  Call Extruder(68.03550)
  MoveL 3349 to (-35.61, 39.11, 59.84) mm, rotated rx -180 ry 0 rz 180 deg; joints [-168.693, 58.392, -72.558, 168.348, 76.115, 2.833]
  MoveL 3350 to (-35.61, 39.11, 59.84) mm, rotated rx -180 ry 0 rz 180 deg; joints [-168.693, 58.392, -72.558, 168.348, 76.115, 2.833]
  Call Extruder(68.23307)
  MoveL 3351 to (-35.35, 38.9, 59.84) mm, rotated rx -180 ry 0 rz 180 deg; joints [-168.739, 58.372, -72.572, 168.394, 76.079, 2.829]
  Call Extruder(68.56709)
  MoveL 3352 to (-34.9, 38.57, 59.84) mm, rotated rx -180 ry 0 rz -180 deg; joints [-168.806, 58.336, -72.595, 168.46, 76.017, 2.824]
  MoveL 3353 to (-34.9, 38.57, 59.84) mm, rotated rx -180 ry 0 rz -180 deg; joints [-168.806, 58.336, -72.595, 168.46, 76.017, 2.824]
  Call Extruder(68.89992)
  MoveL 3354 to (-34.45, 38.24, 59.84) mm, rotated rx -180 ry 0 rz -180 deg; joints [-168.874, 58.3, -72.619, 168.527, 75.955, 2.82]
  MoveL 3355 to (-34.45, 38.24, 59.84) mm, rotated rx -180 ry 0 rz -180 deg; joints [-168.874, 58.3, -72.619, 168.527, 75.955, 2.82]
  Call Extruder(69.07917)
  MoveL 3356 to (-34.21, 38.06, 59.84) mm, rotated rx -180 ry 0 rz 180 deg; joints [-168.91, 58.28, -72.632, 168.562, 75.922, 2.817]
  MoveL 3357 to (-34.21, 38.06, 59.84) mm, rotated rx -180 ry 0 rz 180 deg; joints [-168.91, 58.28, -72.632, 168.562, 75.922, 2.817]
  Call Extruder(69.28728)
  MoveL 3358 to (-33.9, 37.89, 59.84) mm, rotated rx -180 ry 0 rz 180 deg; joints [-168.944, 58.257, -72.647, 168.595, 75.882, 2.817]
  MoveL 3359 to (-33.9, 37.89, 59.84) mm, rotated rx -180 ry 0 rz 180 deg; joints [-168.944, 58.257, -72.647, 168.595, 75.882, 2.817]
  Call Extruder(69.49461)
  MoveL 3360 to (-33.6, 37.71, 59.84) mm, rotated rx 180 ry 0 rz -180 deg; joints [-168.977, 58.233, -72.663, 168.627, 75.842, 2.817]
  MoveL 3361 to (-33.6, 37.71, 59.84) mm, rotated rx 180 ry 0 rz -180 deg; joints [-168.977, 58.233, -72.663, 168.627, 75.842, 2.817]
  Call Extruder(69.70116)
  MoveL 3362 to (-33.29, 37.54, 59.84) mm, rotated rx -180 ry 0 rz -180 deg; joints [-169.01, 58.209, -72.678, 168.659, 75.802, 2.816]
  MoveL 3363 to (-33.29, 37.54, 59.84) mm, rotated rx -180 ry 0 rz -180 deg; joints [-169.01, 58.209, -72.678, 168.659, 75.802, 2.816]
  Call Extruder(69.90693)
  MoveL 3364 to (-32.99, 37.36, 59.84) mm, rotated rx 180 ry 0 rz -180 deg; joints [-169.043, 58.186, -72.694, 168.691, 75.762, 2.816]
  MoveL 3365 to (-32.99, 37.36, 59.84) mm, rotated rx 180 ry 0 rz -180 deg; joints [-169.043, 58.186, -72.694, 168.691, 75.762, 2.816]
  Call Extruder(70.06523)
  MoveL 3366 to (-32.74, 37.26, 59.84) mm, rotated rx -180 ry 0 rz 180 deg; joints [-169.06, 58.167, -72.706, 168.707, 75.731, 2.818]
  MoveL 3367 to (-32.74, 37.26, 59.84) mm, rotated rx -180 ry 0 rz 180 deg; joints [-169.06, 58.167, -72.706, 168.707, 75.731, 2.818]
  Call Extruder(70.22293)
  MoveL 3368 to (-32.49, 37.15, 59.84) mm, rotated rx 180 ry 0 rz 180 deg; joints [-169.077, 58.148, -72.718, 168.723, 75.699, 2.82]
  MoveL 3369 to (-32.49, 37.15, 59.84) mm, rotated rx 180 ry 0 rz 180 deg; joints [-169.077, 58.148, -72.718, 168.723, 75.699, 2.82]
  Call Extruder(70.39301)
  MoveL 3370 to (-32.22, 37.04, 59.84) mm, rotated rx 180 ry 0 rz 180 deg; joints [-169.095, 58.127, -72.731, 168.74, 75.665, 2.822]
  MoveL 3371 to (-32.22, 37.04, 59.84) mm, rotated rx 180 ry 0 rz 180 deg; joints [-169.095, 58.127, -72.731, 168.74, 75.665, 2.822]
  Call Extruder(70.57535)
  MoveL 3372 to (-31.93, 36.91, 59.84) mm, rotated rx -180 ry 0 rz 180 deg; joints [-169.113, 58.105, -72.745, 168.757, 75.629, 2.825]
  MoveL 3373 to (-31.93, 36.91, 59.84) mm, rotated rx -180 ry 0 rz 180 deg; joints [-169.113, 58.105, -72.745, 168.757, 75.629, 2.825]
  Call Extruder(70.75693)
  MoveL 3374 to (-31.64, 36.79, 59.84) mm, rotated rx 180 ry 0 rz -180 deg; joints [-169.132, 58.082, -72.76, 168.774, 75.592, 2.827]
  MoveL 3375 to (-31.64, 36.79, 59.84) mm, rotated rx 180 ry 0 rz -180 deg; joints [-169.132, 58.082, -72.76, 168.774, 75.592, 2.827]
  Call Extruder(70.85628)
  MoveL 3376 to (-31.47, 36.74, 59.84) mm, rotated rx -180 ry 0 rz 180 deg; joints [-169.138, 58.07, -72.767, 168.78, 75.572, 2.83]
  MoveL 3377 to (-31.47, 36.74, 59.84) mm, rotated rx -180 ry 0 rz 180 deg; joints [-169.138, 58.07, -72.767, 168.78, 75.572, 2.83]
  Call Extruder(70.95529)
  MoveL 3378 to (-31.31, 36.69, 59.84) mm, rotated rx -180 ry 0 rz -180 deg; joints [-169.144, 58.058, -72.775, 168.785, 75.552, 2.832]
  MoveL 3379 to (-31.31, 36.69, 59.84) mm, rotated rx -180 ry 0 rz -180 deg; joints [-169.144, 58.058, -72.775, 168.785, 75.552, 2.832]
  Call Extruder(71.05746)
  MoveL 3380 to (-31.14, 36.63, 59.84) mm, rotated rx -180 ry 0 rz -180 deg; joints [-169.151, 58.045, -72.783, 168.791, 75.531, 2.835]
  MoveL 3381 to (-31.14, 36.63, 59.84) mm, rotated rx -180 ry 0 rz -180 deg; joints [-169.151, 58.045, -72.783, 168.791, 75.531, 2.835]
  Call Extruder(71.16269)
  MoveL 3382 to (-30.96, 36.57, 59.84) mm, rotated rx 180 ry 0 rz 180 deg; joints [-169.158, 58.032, -72.792, 168.797, 75.509, 2.837]
  MoveL 3383 to (-30.96, 36.57, 59.84) mm, rotated rx 180 ry 0 rz 180 deg; joints [-169.158, 58.032, -72.792, 168.797, 75.509, 2.837]
  Call Extruder(71.26752)
  MoveL 3384 to (-30.78, 36.52, 59.84) mm, rotated rx -180 ry 0 rz 180 deg; joints [-169.165, 58.018, -72.8, 168.803, 75.488, 2.84]
  MoveL 3385 to (-30.78, 36.52, 59.84) mm, rotated rx -180 ry 0 rz 180 deg; joints [-169.165, 58.018, -72.8, 168.803, 75.488, 2.84]
  Call Extruder(71.38542)
  MoveL 3386 to (-30.58, 36.45, 59.84) mm, rotated rx 180 ry 0 rz -180 deg; joints [-169.172, 58.003, -72.809, 168.809, 75.463, 2.843]
  MoveL 3387 to (-30.58, 36.45, 59.84) mm, rotated rx 180 ry 0 rz -180 deg; joints [-169.172, 58.003, -72.809, 168.809, 75.463, 2.843]
  Call Extruder(71.51620)
  MoveL 3388 to (-30.36, 36.38, 59.84) mm, rotated rx 180 ry 0 rz 180 deg; joints [-169.179, 57.986, -72.82, 168.815, 75.436, 2.846]
  MoveL 3389 to (-30.36, 36.38, 59.84) mm, rotated rx 180 ry 0 rz 180 deg; joints [-169.179, 57.986, -72.82, 168.815, 75.436, 2.846]
  Call Extruder(71.64643)
  MoveL 3390 to (-30.14, 36.32, 59.84) mm, rotated rx 180 ry 0 rz 180 deg; joints [-169.186, 57.97, -72.83, 168.821, 75.409, 2.85]
  MoveL 3391 to (-30.14, 36.32, 59.84) mm, rotated rx 180 ry 0 rz 180 deg; joints [-169.186, 57.97, -72.83, 168.821, 75.409, 2.85]
  Call Extruder(71.77608)
  MoveL 3392 to (-29.91, 36.25, 59.84) mm, rotated rx -180 ry 0 rz -180 deg; joints [-169.193, 57.953, -72.841, 168.827, 75.382, 2.854]
  MoveL 3393 to (-29.91, 36.25, 59.84) mm, rotated rx -180 ry 0 rz -180 deg; joints [-169.193, 57.953, -72.841, 168.827, 75.382, 2.854]
  Call Extruder(71.90518)
  MoveL 3394 to (-29.69, 36.18, 59.84) mm, rotated rx -180 ry 0 rz -180 deg; joints [-169.201, 57.936, -72.851, 168.833, 75.355, 2.857]
  MoveL 3395 to (-29.69, 36.18, 59.84) mm, rotated rx -180 ry 0 rz -180 deg; joints [-169.201, 57.936, -72.851, 168.833, 75.355, 2.857]
  Call Extruder(72.02025)
  MoveL 3396 to (-29.48, 36.14, 59.84) mm, rotated rx -180 ry 0 rz 180 deg; joints [-169.202, 57.921, -72.861, 168.834, 75.33, 2.862]
  MoveL 3397 to (-29.48, 36.14, 59.84) mm, rotated rx -180 ry 0 rz 180 deg; joints [-169.202, 57.921, -72.861, 168.834, 75.33, 2.862]
  Call Extruder(72.13487)
  MoveL 3398 to (-29.28, 36.09, 59.84) mm, rotated rx -180 ry 0 rz -180 deg; joints [-169.204, 57.905, -72.87, 168.834, 75.306, 2.866]
  MoveL 3399 to (-29.28, 36.09, 59.84) mm, rotated rx -180 ry 0 rz -180 deg; joints [-169.204, 57.905, -72.87, 168.834, 75.306, 2.866]
  Call Extruder(72.24904)
  MoveL 3400 to (-29.08, 36.05, 59.84) mm, rotated rx -180 ry 0 rz 180 deg; joints [-169.206, 57.89, -72.879, 168.835, 75.282, 2.871]
  MoveL 3401 to (-29.08, 36.05, 59.84) mm, rotated rx -180 ry 0 rz 180 deg; joints [-169.206, 57.89, -72.879, 168.835, 75.282, 2.871]
  Call Extruder(72.36276)
  MoveL 3402 to (-28.87, 36, 59.84) mm, rotated rx -180 ry 0 rz -180 deg; joints [-169.207, 57.875, -72.889, 168.835, 75.258, 2.875]
  MoveL 3403 to (-28.87, 36, 59.84) mm, rotated rx -180 ry 0 rz -180 deg; joints [-169.207, 57.875, -72.889, 168.835, 75.258, 2.875]
  Call Extruder(72.48818)
  MoveL 3404 to (-28.65, 35.96, 59.84) mm, rotated rx -180 ry 0 rz -180 deg; joints [-169.208, 57.858, -72.899, 168.835, 75.231, 2.88]
  MoveL 3405 to (-28.65, 35.96, 59.84) mm, rotated rx -180 ry 0 rz -180 deg; joints [-169.208, 57.858, -72.899, 168.835, 75.231, 2.88]
  Call Extruder(72.62516)
  MoveL 3406 to (-28.4, 35.91, 59.84) mm, rotated rx -180 ry 0 rz 180 deg; joints [-169.209, 57.84, -72.91, 168.834, 75.202, 2.886]
  MoveL 3407 to (-28.4, 35.91, 59.84) mm, rotated rx -180 ry 0 rz 180 deg; joints [-169.209, 57.84, -72.91, 168.834, 75.202, 2.886]
  Call Extruder(72.76152)
  MoveL 3408 to (-28.15, 35.86, 59.84) mm, rotated rx -180 ry 0 rz -180 deg; joints [-169.21, 57.821, -72.921, 168.833, 75.173, 2.892]
  MoveL 3409 to (-28.15, 35.86, 59.84) mm, rotated rx -180 ry 0 rz -180 deg; joints [-169.21, 57.821, -72.921, 168.833, 75.173, 2.892]
  Call Extruder(72.89728)
  MoveL 3410 to (-27.9, 35.81, 59.84) mm, rotated rx 180 ry 0 rz 180 deg; joints [-169.21, 57.803, -72.933, 168.833, 75.144, 2.898]
  MoveL 3411 to (-27.9, 35.81, 59.84) mm, rotated rx 180 ry 0 rz 180 deg; joints [-169.21, 57.803, -72.933, 168.833, 75.144, 2.898]
  Call Extruder(73.03243)
  MoveL 3412 to (-27.65, 35.76, 59.84) mm, rotated rx -180 ry 0 rz -180 deg; joints [-169.211, 57.784, -72.944, 168.831, 75.114, 2.904]
  MoveL 3413 to (-27.65, 35.76, 59.84) mm, rotated rx -180 ry 0 rz -180 deg; joints [-169.211, 57.784, -72.944, 168.831, 75.114, 2.904]
  Call Extruder(73.16696)
  MoveL 3414 to (-27.4, 35.71, 59.84) mm, rotated rx -180 ry 0 rz 180 deg; joints [-169.212, 57.765, -72.955, 168.831, 75.085, 2.909]
  MoveL 3415 to (-27.4, 35.71, 59.84) mm, rotated rx -180 ry 0 rz 180 deg; joints [-169.212, 57.765, -72.955, 168.831, 75.085, 2.909]
  Call Extruder(73.30089)
  MoveL 3416 to (-27.15, 35.66, 59.84) mm, rotated rx 180 ry 0 rz 180 deg; joints [-169.212, 57.747, -72.966, 168.83, 75.056, 2.915]
  MoveL 3417 to (-27.15, 35.66, 59.84) mm, rotated rx 180 ry 0 rz 180 deg; joints [-169.212, 57.747, -72.966, 168.83, 75.056, 2.915]
  Call Extruder(73.44875)
  MoveL 3418 to (-26.87, 35.61, 59.84) mm, rotated rx -180 ry 0 rz 180 deg; joints [-169.211, 57.726, -72.978, 168.827, 75.024, 2.922]
  MoveL 3419 to (-26.87, 35.61, 59.84) mm, rotated rx -180 ry 0 rz 180 deg; joints [-169.211, 57.726, -72.978, 168.827, 75.024, 2.922]
  Call Extruder(73.61048)
  MoveL 3420 to (-26.57, 35.56, 59.84) mm, rotated rx 180 ry 0 rz 180 deg; joints [-169.208, 57.703, -72.992, 168.822, 74.988, 2.93]
  MoveL 3421 to (-26.57, 35.56, 59.84) mm, rotated rx 180 ry 0 rz 180 deg; joints [-169.208, 57.703, -72.992, 168.822, 74.988, 2.93]
  Call Extruder(73.77149)
  MoveL 3422 to (-26.26, 35.51, 59.84) mm, rotated rx -180 ry 0 rz -180 deg; joints [-169.205, 57.681, -73.006, 168.817, 74.953, 2.938]
  MoveL 3423 to (-26.26, 35.51, 59.84) mm, rotated rx -180 ry 0 rz -180 deg; joints [-169.205, 57.681, -73.006, 168.817, 74.953, 2.938]
  Call Extruder(73.93177)
  MoveL 3424 to (-25.96, 35.46, 59.84) mm, rotated rx 180 ry 0 rz 180 deg; joints [-169.202, 57.658, -73.019, 168.812, 74.917, 2.946]
  MoveL 3425 to (-25.96, 35.46, 59.84) mm, rotated rx 180 ry 0 rz 180 deg; joints [-169.202, 57.658, -73.019, 168.812, 74.917, 2.946]
  Call Extruder(74.09132)
  MoveL 3426 to (-25.65, 35.42, 59.84) mm, rotated rx 180 ry 0 rz 180 deg; joints [-169.199, 57.635, -73.032, 168.807, 74.882, 2.954]
  MoveL 3427 to (-25.65, 35.42, 59.84) mm, rotated rx 180 ry 0 rz 180 deg; joints [-169.199, 57.635, -73.032, 168.807, 74.882, 2.954]
  Call Extruder(74.25014)
  MoveL 3428 to (-25.34, 35.37, 59.84) mm, rotated rx -180 ry 0 rz 180 deg; joints [-169.196, 57.612, -73.046, 168.802, 74.847, 2.962]
  MoveL 3429 to (-25.34, 35.37, 59.84) mm, rotated rx -180 ry 0 rz 180 deg; joints [-169.196, 57.612, -73.046, 168.802, 74.847, 2.962]
  Call Extruder(74.42881)
  MoveL 3430 to (-25, 35.32, 59.84) mm, rotated rx 180 ry 0 rz 180 deg; joints [-169.191, 57.586, -73.061, 168.794, 74.807, 2.972]
  MoveL 3431 to (-25, 35.32, 59.84) mm, rotated rx 180 ry 0 rz 180 deg; joints [-169.191, 57.586, -73.061, 168.794, 74.807, 2.972]
  Call Extruder(74.62725)
  MoveL 3432 to (-24.61, 35.28, 59.84) mm, rotated rx 180 ry 0 rz -180 deg; joints [-169.182, 57.558, -73.077, 168.783, 74.763, 2.984]
  MoveL 3433 to (-24.61, 35.28, 59.84) mm, rotated rx 180 ry 0 rz -180 deg; joints [-169.182, 57.558, -73.077, 168.783, 74.763, 2.984]
  Call Extruder(74.82483)
  MoveL 3434 to (-24.22, 35.23, 59.84) mm, rotated rx -180 ry 0 rz -180 deg; joints [-169.174, 57.529, -73.094, 168.772, 74.719, 2.995]
  MoveL 3435 to (-24.22, 35.23, 59.84) mm, rotated rx -180 ry 0 rz -180 deg; joints [-169.174, 57.529, -73.094, 168.772, 74.719, 2.995]
  Call Extruder(75.02153)
  MoveL 3436 to (-23.84, 35.18, 59.84) mm, rotated rx -180 ry 0 rz 180 deg; joints [-169.166, 57.5, -73.111, 168.761, 74.674, 3.006]
  MoveL 3437 to (-23.84, 35.18, 59.84) mm, rotated rx -180 ry 0 rz 180 deg; joints [-169.166, 57.5, -73.111, 168.761, 74.674, 3.006]
  Call Extruder(75.21737)
  MoveL 3438 to (-23.45, 35.14, 59.84) mm, rotated rx 180 ry 0 rz -180 deg; joints [-169.157, 57.471, -73.127, 168.749, 74.63, 3.018]
  MoveL 3439 to (-23.45, 35.14, 59.84) mm, rotated rx 180 ry 0 rz -180 deg; joints [-169.157, 57.471, -73.127, 168.749, 74.63, 3.018]
  Call Extruder(75.51277)
  MoveL 3440 to (-22.86, 35.09, 59.84) mm, rotated rx -180 ry 0 rz 180 deg; joints [-169.137, 57.427, -73.152, 168.725, 74.564, 3.037]
  MoveL 3441 to (-22.86, 35.09, 59.84) mm, rotated rx -180 ry 0 rz 180 deg; joints [-169.137, 57.427, -73.152, 168.725, 74.564, 3.037]
  Call Extruder(75.80683)
  MoveL 3442 to (-22.27, 35.05, 59.84) mm, rotated rx -180 ry 0 rz -180 deg; joints [-169.117, 57.383, -73.177, 168.7, 74.498, 3.057]
  MoveL 3443 to (-22.27, 35.05, 59.84) mm, rotated rx -180 ry 0 rz -180 deg; joints [-169.117, 57.383, -73.177, 168.7, 74.498, 3.057]
  Call Extruder(76.09956)
  MoveL 3444 to (-21.68, 35, 59.84) mm, rotated rx 180 ry 0 rz 180 deg; joints [-169.096, 57.339, -73.201, 168.676, 74.432, 3.077]
  MoveL 3445 to (-21.68, 35, 59.84) mm, rotated rx 180 ry 0 rz 180 deg; joints [-169.096, 57.339, -73.201, 168.676, 74.432, 3.077]
  Call Extruder(76.67301)
  MoveL 3446 to (-20.52, 34.95, 59.84) mm, rotated rx -180 ry 0 rz -180 deg; joints [-169.042, 57.253, -73.249, 168.612, 74.303, 3.119]
  MoveL 3447 to (-20.52, 34.95, 59.84) mm, rotated rx -180 ry 0 rz -180 deg; joints [-169.042, 57.253, -73.249, 168.612, 74.303, 3.119]
  Call Extruder(77.38698)
  MoveL 3448 to (-19.06, 34.91, 59.84) mm, rotated rx 180 ry 0 rz 180 deg; joints [-168.967, 57.145, -73.308, 168.525, 74.144, 3.175]
  Call Extruder(194.23372)
  MoveL 3449 to (219.06, 34.91, 59.84) mm, rotated rx 180 ry 0 rz 180 deg; joints [-30.588, 46.892, -75.487, 33.95, 114.332, 15.503]
  Call Extruder(194.66228)
  MoveL 3450 to (219.94, 34.93, 59.84) mm, rotated rx 180 ry 0 rz 180 deg; joints [-30.233, 46.97, -75.489, 33.555, 114.362, 15.302]
  MoveL 3451 to (219.94, 34.93, 59.84) mm, rotated rx 180 ry 0 rz 180 deg; joints [-30.233, 46.97, -75.489, 33.555, 114.362, 15.302]
  Call Extruder(195.23572)
  MoveL 3452 to (221.1, 34.98, 59.84) mm, rotated rx -180 ry 0 rz 180 deg; joints [-29.789, 47.076, -75.491, 33.058, 114.392, 15.044]
  MoveL 3453 to (221.1, 34.98, 59.84) mm, rotated rx -180 ry 0 rz 180 deg; joints [-29.789, 47.076, -75.491, 33.058, 114.392, 15.044]
  Call Extruder(195.67004)
  MoveL 3454 to (221.97, 35.02, 59.84) mm, rotated rx 180 ry 0 rz 180 deg; joints [-29.47, 47.157, -75.492, 32.701, 114.407, 14.858]
  MoveL 3455 to (221.97, 35.02, 59.84) mm, rotated rx 180 ry 0 rz 180 deg; joints [-29.47, 47.157, -75.492, 32.701, 114.407, 14.858]
  Call Extruder(195.96409)
  MoveL 3456 to (222.56, 35.07, 59.84) mm, rotated rx -180 ry 0 rz -180 deg; joints [-29.272, 47.212, -75.493, 32.477, 114.412, 14.738]
  MoveL 3457 to (222.56, 35.07, 59.84) mm, rotated rx -180 ry 0 rz -180 deg; joints [-29.272, 47.212, -75.493, 32.477, 114.412, 14.738]
  Call Extruder(196.25948)
  MoveL 3458 to (223.15, 35.11, 59.84) mm, rotated rx 180 ry 0 rz 180 deg; joints [-29.075, 47.267, -75.493, 32.254, 114.416, 14.62]
  MoveL 3459 to (223.15, 35.11, 59.84) mm, rotated rx 180 ry 0 rz 180 deg; joints [-29.075, 47.267, -75.493, 32.254, 114.416, 14.62]
  Call Extruder(196.50572)
  MoveL 3460 to (223.64, 35.16, 59.84) mm, rotated rx 180 ry 0 rz 180 deg; joints [-28.92, 47.313, -75.494, 32.078, 114.416, 14.525]
  MoveL 3461 to (223.64, 35.16, 59.84) mm, rotated rx 180 ry 0 rz 180 deg; joints [-28.92, 47.313, -75.494, 32.078, 114.416, 14.525]
  Call Extruder(196.70242)
  MoveL 3462 to (224.03, 35.21, 59.84) mm, rotated rx 180 ry 0 rz 180 deg; joints [-28.804, 47.35, -75.494, 31.946, 114.414, 14.453]
  MoveL 3463 to (224.03, 35.21, 59.84) mm, rotated rx 180 ry 0 rz 180 deg; joints [-28.804, 47.35, -75.494, 31.946, 114.414, 14.453]
  Call Extruder(196.90000)
  MoveL 3464 to (224.42, 35.25, 59.84) mm, rotated rx -180 ry 0 rz 180 deg; joints [-28.69, 47.387, -75.494, 31.816, 114.411, 14.381]
  MoveL 3465 to (224.42, 35.25, 59.84) mm, rotated rx -180 ry 0 rz 180 deg; joints [-28.69, 47.387, -75.494, 31.816, 114.411, 14.381]
  Call Extruder(197.09844)
  MoveL 3466 to (224.8, 35.3, 59.84) mm, rotated rx -180 ry 0 rz 180 deg; joints [-28.577, 47.424, -75.495, 31.687, 114.408, 14.31]
  MoveL 3467 to (224.8, 35.3, 59.84) mm, rotated rx -180 ry 0 rz 180 deg; joints [-28.577, 47.424, -75.495, 31.687, 114.408, 14.31]
  Call Extruder(197.29775)
  MoveL 3468 to (225.19, 35.34, 59.84) mm, rotated rx -180 ry 0 rz 180 deg; joints [-28.465, 47.461, -75.495, 31.559, 114.404, 14.24]
  MoveL 3469 to (225.19, 35.34, 59.84) mm, rotated rx -180 ry 0 rz 180 deg; joints [-28.465, 47.461, -75.495, 31.559, 114.404, 14.24]
  Call Extruder(197.45657)
  MoveL 3470 to (225.5, 35.39, 59.84) mm, rotated rx 180 ry 0 rz 180 deg; joints [-28.385, 47.491, -75.495, 31.467, 114.398, 14.188]
  MoveL 3471 to (225.5, 35.39, 59.84) mm, rotated rx 180 ry 0 rz 180 deg; joints [-28.385, 47.491, -75.495, 31.467, 114.398, 14.188]
  Call Extruder(197.61612)
  MoveL 3472 to (225.8, 35.44, 59.84) mm, rotated rx -180 ry 0 rz 180 deg; joints [-28.307, 47.521, -75.495, 31.377, 114.392, 14.136]
  MoveL 3473 to (225.8, 35.44, 59.84) mm, rotated rx -180 ry 0 rz 180 deg; joints [-28.307, 47.521, -75.495, 31.377, 114.392, 14.136]
  Call Extruder(197.77640)
  MoveL 3474 to (226.11, 35.49, 59.84) mm, rotated rx 180 ry 0 rz 180 deg; joints [-28.228, 47.551, -75.495, 31.286, 114.386, 14.085]
  MoveL 3475 to (226.11, 35.49, 59.84) mm, rotated rx 180 ry 0 rz 180 deg; joints [-28.228, 47.551, -75.495, 31.286, 114.386, 14.085]
  Call Extruder(197.93740)
  MoveL 3476 to (226.41, 35.54, 59.84) mm, rotated rx 180 ry 0 rz 180 deg; joints [-28.151, 47.581, -75.495, 31.197, 114.379, 14.034]
  MoveL 3477 to (226.41, 35.54, 59.84) mm, rotated rx 180 ry 0 rz 180 deg; joints [-28.151, 47.581, -75.495, 31.197, 114.379, 14.034]
  Call Extruder(198.09914)
  MoveL 3478 to (226.72, 35.59, 59.84) mm, rotated rx -180 ry 0 rz 180 deg; joints [-28.074, 47.61, -75.495, 31.108, 114.372, 13.983]
  MoveL 3479 to (226.72, 35.59, 59.84) mm, rotated rx -180 ry 0 rz 180 deg; joints [-28.074, 47.61, -75.495, 31.108, 114.372, 13.983]
  Call Extruder(198.26160)
  MoveL 3480 to (227.02, 35.63, 59.84) mm, rotated rx -180 ry 0 rz 180 deg; joints [-27.998, 47.64, -75.495, 31.02, 114.365, 13.933]
  MoveL 3481 to (227.02, 35.63, 59.84) mm, rotated rx -180 ry 0 rz 180 deg; joints [-27.998, 47.64, -75.495, 31.02, 114.365, 13.933]
  Call Extruder(198.39552)
  MoveL 3482 to (227.28, 35.68, 59.84) mm, rotated rx -180 ry 0 rz 180 deg; joints [-27.942, 47.665, -75.495, 30.955, 114.357, 13.894]
  MoveL 3483 to (227.28, 35.68, 59.84) mm, rotated rx -180 ry 0 rz 180 deg; joints [-27.942, 47.665, -75.495, 30.955, 114.357, 13.894]
  Call Extruder(198.53006)
  MoveL 3484 to (227.52, 35.73, 59.84) mm, rotated rx -180 ry 0 rz 180 deg; joints [-27.888, 47.69, -75.495, 30.891, 114.349, 13.856]
  MoveL 3485 to (227.52, 35.73, 59.84) mm, rotated rx -180 ry 0 rz 180 deg; joints [-27.888, 47.69, -75.495, 30.891, 114.349, 13.856]
  Call Extruder(198.66521)
  MoveL 3486 to (227.77, 35.78, 59.84) mm, rotated rx -180 ry 0 rz 180 deg; joints [-27.834, 47.715, -75.494, 30.828, 114.34, 13.818]
  MoveL 3487 to (227.77, 35.78, 59.84) mm, rotated rx -180 ry 0 rz 180 deg; joints [-27.834, 47.715, -75.494, 30.828, 114.34, 13.818]
  Call Extruder(198.80097)
  MoveL 3488 to (228.02, 35.83, 59.84) mm, rotated rx -180 ry 0 rz -180 deg; joints [-27.78, 47.739, -75.494, 30.764, 114.332, 13.781]
  MoveL 3489 to (228.02, 35.83, 59.84) mm, rotated rx -180 ry 0 rz -180 deg; joints [-27.78, 47.739, -75.494, 30.764, 114.332, 13.781]
  Call Extruder(198.93734)
  MoveL 3490 to (228.27, 35.88, 59.84) mm, rotated rx -180 ry 0 rz 180 deg; joints [-27.726, 47.764, -75.494, 30.702, 114.323, 13.743]
  MoveL 3491 to (228.27, 35.88, 59.84) mm, rotated rx -180 ry 0 rz 180 deg; joints [-27.726, 47.764, -75.494, 30.702, 114.323, 13.743]
  Call Extruder(199.07431)
  MoveL 3492 to (228.52, 35.93, 59.84) mm, rotated rx 180 ry 0 rz 180 deg; joints [-27.673, 47.789, -75.494, 30.639, 114.314, 13.706]
  MoveL 3493 to (228.52, 35.93, 59.84) mm, rotated rx 180 ry 0 rz 180 deg; joints [-27.673, 47.789, -75.494, 30.639, 114.314, 13.706]
  Call Extruder(199.21190)
  MoveL 3494 to (228.77, 35.98, 59.84) mm, rotated rx 180 ry 0 rz -180 deg; joints [-27.62, 47.813, -75.494, 30.577, 114.305, 13.669]
  MoveL 3495 to (228.77, 35.98, 59.84) mm, rotated rx 180 ry 0 rz -180 deg; joints [-27.62, 47.813, -75.494, 30.577, 114.305, 13.669]
  Call Extruder(199.32562)
  MoveL 3496 to (228.97, 36.03, 59.84) mm, rotated rx -180 ry 0 rz 180 deg; joints [-27.579, 47.834, -75.493, 30.528, 114.297, 13.639]
  MoveL 3497 to (228.97, 36.03, 59.84) mm, rotated rx -180 ry 0 rz 180 deg; joints [-27.579, 47.834, -75.493, 30.528, 114.297, 13.639]
  Call Extruder(199.43979)
  MoveL 3498 to (229.18, 36.07, 59.84) mm, rotated rx 180 ry 0 rz 180 deg; joints [-27.539, 47.854, -75.493, 30.481, 114.289, 13.61]
  MoveL 3499 to (229.18, 36.07, 59.84) mm, rotated rx 180 ry 0 rz 180 deg; joints [-27.539, 47.854, -75.493, 30.481, 114.289, 13.61]
  Call Extruder(199.55441)
  MoveL 3500 to (229.38, 36.12, 59.84) mm, rotated rx -180 ry 0 rz 180 deg; joints [-27.499, 47.875, -75.493, 30.433, 114.28, 13.581]
  MoveL 3501 to (229.38, 36.12, 59.84) mm, rotated rx -180 ry 0 rz 180 deg; joints [-27.499, 47.875, -75.493, 30.433, 114.28, 13.581]
  Call Extruder(199.66948)
  MoveL 3502 to (229.59, 36.16, 59.84) mm, rotated rx -180 ry 0 rz 180 deg; joints [-27.458, 47.895, -75.493, 30.386, 114.272, 13.552]
  MoveL 3503 to (229.59, 36.16, 59.84) mm, rotated rx -180 ry 0 rz 180 deg; joints [-27.458, 47.895, -75.493, 30.386, 114.272, 13.552]
  Call Extruder(199.79172)
  MoveL 3504 to (229.8, 36.22, 59.84) mm, rotated rx -180 ry 0 rz 180 deg; joints [-27.423, 47.917, -75.492, 30.343, 114.261, 13.524]
  MoveL 3505 to (229.8, 36.22, 59.84) mm, rotated rx -180 ry 0 rz 180 deg; joints [-27.423, 47.917, -75.492, 30.343, 114.261, 13.524]
  Call Extruder(199.92138)
  MoveL 3506 to (230.02, 36.28, 59.84) mm, rotated rx 180 ry 0 rz -180 deg; joints [-27.392, 47.94, -75.492, 30.304, 114.248, 13.497]
  MoveL 3507 to (230.02, 36.28, 59.84) mm, rotated rx 180 ry 0 rz -180 deg; joints [-27.392, 47.94, -75.492, 30.304, 114.248, 13.497]
  Call Extruder(200.05161)
  MoveL 3508 to (230.25, 36.35, 59.84) mm, rotated rx -180 ry 0 rz 180 deg; joints [-27.361, 47.963, -75.492, 30.266, 114.235, 13.471]
  MoveL 3509 to (230.25, 36.35, 59.84) mm, rotated rx -180 ry 0 rz 180 deg; joints [-27.361, 47.963, -75.492, 30.266, 114.235, 13.471]
  Call Extruder(200.18241)
  MoveL 3510 to (230.47, 36.42, 59.84) mm, rotated rx 180 ry 0 rz -180 deg; joints [-27.33, 47.987, -75.491, 30.227, 114.222, 13.444]
  MoveL 3511 to (230.47, 36.42, 59.84) mm, rotated rx 180 ry 0 rz -180 deg; joints [-27.33, 47.987, -75.491, 30.227, 114.222, 13.444]
  Call Extruder(200.31377)
  MoveL 3512 to (230.69, 36.49, 59.84) mm, rotated rx -180 ry 0 rz 180 deg; joints [-27.299, 48.01, -75.491, 30.189, 114.209, 13.418]
  MoveL 3513 to (230.69, 36.49, 59.84) mm, rotated rx -180 ry 0 rz 180 deg; joints [-27.299, 48.01, -75.491, 30.189, 114.209, 13.418]
  Call Extruder(200.43194)
  MoveL 3514 to (230.89, 36.55, 59.84) mm, rotated rx -180 ry 0 rz 180 deg; joints [-27.275, 48.031, -75.491, 30.159, 114.196, 13.395]
  MoveL 3515 to (230.89, 36.55, 59.84) mm, rotated rx -180 ry 0 rz 180 deg; joints [-27.275, 48.031, -75.491, 30.159, 114.196, 13.395]
  Call Extruder(200.55059)
  MoveL 3516 to (231.09, 36.62, 59.84) mm, rotated rx -180 ry 0 rz 180 deg; joints [-27.25, 48.052, -75.49, 30.128, 114.183, 13.373]
  MoveL 3517 to (231.09, 36.62, 59.84) mm, rotated rx -180 ry 0 rz 180 deg; joints [-27.25, 48.052, -75.49, 30.128, 114.183, 13.373]
  Call Extruder(200.66975)
  MoveL 3518 to (231.29, 36.68, 59.84) mm, rotated rx 180 ry 0 rz 180 deg; joints [-27.227, 48.072, -75.49, 30.098, 114.17, 13.351]
  MoveL 3519 to (231.29, 36.68, 59.84) mm, rotated rx 180 ry 0 rz 180 deg; joints [-27.227, 48.072, -75.49, 30.098, 114.17, 13.351]
  Call Extruder(200.77883)
  MoveL 3520 to (231.47, 36.74, 59.84) mm, rotated rx 180 ry 0 rz 180 deg; joints [-27.205, 48.091, -75.489, 30.07, 114.159, 13.331]
  MoveL 3521 to (231.47, 36.74, 59.84) mm, rotated rx 180 ry 0 rz 180 deg; joints [-27.205, 48.091, -75.489, 30.07, 114.159, 13.331]
  Call Extruder(200.87772)
  MoveL 3522 to (231.64, 36.79, 59.84) mm, rotated rx -180 ry 0 rz 180 deg; joints [-27.185, 48.108, -75.489, 30.045, 114.148, 13.313]
  MoveL 3523 to (231.64, 36.79, 59.84) mm, rotated rx -180 ry 0 rz 180 deg; joints [-27.185, 48.108, -75.489, 30.045, 114.148, 13.313]
  Call Extruder(201.05968)
  MoveL 3524 to (231.93, 36.91, 59.84) mm, rotated rx -180 ry 0 rz -180 deg; joints [-27.167, 48.14, -75.488, 30.018, 114.124, 13.287]
  MoveL 3525 to (231.93, 36.91, 59.84) mm, rotated rx -180 ry 0 rz -180 deg; joints [-27.167, 48.14, -75.488, 30.018, 114.124, 13.287]
  Call Extruder(201.24239)
  MoveL 3526 to (232.22, 37.03, 59.84) mm, rotated rx 180 ry 0 rz 180 deg; joints [-27.149, 48.172, -75.488, 29.992, 114.1, 13.261]
  MoveL 3527 to (232.22, 37.03, 59.84) mm, rotated rx 180 ry 0 rz 180 deg; joints [-27.149, 48.172, -75.488, 29.992, 114.1, 13.261]
  Call Extruder(201.41281)
  MoveL 3528 to (232.49, 37.15, 59.84) mm, rotated rx -180 ry 0 rz 180 deg; joints [-27.133, 48.201, -75.487, 29.969, 114.078, 13.238]
  MoveL 3529 to (232.49, 37.15, 59.84) mm, rotated rx -180 ry 0 rz 180 deg; joints [-27.133, 48.201, -75.487, 29.969, 114.078, 13.238]
  Call Extruder(201.57081)
  MoveL 3530 to (232.74, 37.26, 59.84) mm, rotated rx -180 ry 0 rz 180 deg; joints [-27.121, 48.229, -75.486, 29.949, 114.057, 13.217]
  MoveL 3531 to (232.74, 37.26, 59.84) mm, rotated rx -180 ry 0 rz 180 deg; joints [-27.121, 48.229, -75.486, 29.949, 114.057, 13.217]
  Call Extruder(201.72941)
  MoveL 3532 to (232.99, 37.36, 59.84) mm, rotated rx -180 ry 0 rz -180 deg; joints [-27.108, 48.256, -75.486, 29.929, 114.035, 13.196]
  MoveL 3533 to (232.99, 37.36, 59.84) mm, rotated rx -180 ry 0 rz -180 deg; joints [-27.108, 48.256, -75.486, 29.929, 114.035, 13.196]
  Call Extruder(201.93558)
  MoveL 3534 to (233.29, 37.54, 59.84) mm, rotated rx -180 ry 0 rz 180 deg; joints [-27.12, 48.291, -75.485, 29.933, 114.001, 13.182]
  MoveL 3535 to (233.29, 37.54, 59.84) mm, rotated rx -180 ry 0 rz 180 deg; joints [-27.12, 48.291, -75.485, 29.933, 114.001, 13.182]
  Call Extruder(202.14252)
  MoveL 3536 to (233.6, 37.71, 59.84) mm, rotated rx 180 ry 0 rz 180 deg; joints [-27.132, 48.326, -75.484, 29.939, 113.967, 13.167]
  MoveL 3537 to (233.6, 37.71, 59.84) mm, rotated rx 180 ry 0 rz 180 deg; joints [-27.132, 48.326, -75.484, 29.939, 113.967, 13.167]
  Call Extruder(202.35025)
  MoveL 3538 to (233.9, 37.89, 59.84) mm, rotated rx 180 ry 0 rz 180 deg; joints [-27.144, 48.361, -75.483, 29.943, 113.933, 13.153]
  MoveL 3539 to (233.9, 37.89, 59.84) mm, rotated rx 180 ry 0 rz 180 deg; joints [-27.144, 48.361, -75.483, 29.943, 113.933, 13.153]
  Call Extruder(202.55875)
  MoveL 3540 to (234.21, 38.07, 59.84) mm, rotated rx 180 ry 0 rz 180 deg; joints [-27.156, 48.396, -75.482, 29.948, 113.899, 13.138]
  MoveL 3541 to (234.21, 38.07, 59.84) mm, rotated rx 180 ry 0 rz 180 deg; joints [-27.156, 48.396, -75.482, 29.948, 113.899, 13.138]
  Call Extruder(202.73829)
  MoveL 3542 to (234.45, 38.24, 59.84) mm, rotated rx -180 ry 0 rz 180 deg; joints [-27.187, 48.426, -75.481, 29.974, 113.865, 13.135]
  MoveL 3543 to (234.45, 38.24, 59.84) mm, rotated rx -180 ry 0 rz 180 deg; joints [-27.187, 48.426, -75.481, 29.974, 113.865, 13.135]
  Call Extruder(203.07171)
  MoveL 3544 to (234.9, 38.57, 59.84) mm, rotated rx 180 ry 0 rz 180 deg; joints [-27.245, 48.481, -75.479, 30.024, 113.803, 13.129]
  MoveL 3545 to (234.9, 38.57, 59.84) mm, rotated rx 180 ry 0 rz 180 deg; joints [-27.245, 48.481, -75.479, 30.024, 113.803, 13.129]
  Call Extruder(203.40631)
  MoveL 3546 to (235.35, 38.9, 59.84) mm, rotated rx 180 ry 0 rz 180 deg; joints [-27.302, 48.537, -75.477, 30.072, 113.74, 13.122]
  Call Extruder(204.23426)
  MoveL 3547 to (236.39, 39.81, 59.84) mm, rotated rx 180 ry 0 rz 180 deg; joints [-27.525, 48.67, -75.471, 30.278, 113.569, 13.141]
  Call Extruder(205.06220)
  MoveL 3548 to (237.3, 40.85, 59.84) mm, rotated rx -180 ry 0 rz 180 deg; joints [-27.851, 48.798, -75.466, 30.595, 113.379, 13.205]
  Call Extruder(205.22950)
  MoveL 3549 to (237.47, 41.07, 59.84) mm, rotated rx -180 ry 0 rz 180 deg; joints [-27.932, 48.823, -75.464, 30.675, 113.339, 13.224]
  MoveL 3550 to (237.47, 41.07, 59.84) mm, rotated rx -180 ry 0 rz 180 deg; joints [-27.932, 48.823, -75.464, 30.675, 113.339, 13.224]
  Call Extruder(205.56292)
  MoveL 3551 to (237.79, 41.52, 59.84) mm, rotated rx -180 ry 0 rz -180 deg; joints [-28.091, 48.873, -75.462, 30.832, 113.257, 13.262]
  MoveL 3552 to (237.79, 41.52, 59.84) mm, rotated rx -180 ry 0 rz -180 deg; joints [-28.091, 48.873, -75.462, 30.832, 113.257, 13.262]
  Call Extruder(205.89514)
  MoveL 3553 to (238.12, 41.97, 59.84) mm, rotated rx -180 ry 0 rz 180 deg; joints [-28.249, 48.923, -75.459, 30.987, 113.176, 13.298]
  MoveL 3554 to (238.12, 41.97, 59.84) mm, rotated rx -180 ry 0 rz 180 deg; joints [-28.249, 48.923, -75.459, 30.987, 113.176, 13.298]
  Call Extruder(206.01284)
  MoveL 3555 to (238.22, 42.15, 59.84) mm, rotated rx -180 ry 0 rz 180 deg; joints [-28.315, 48.939, -75.459, 31.054, 113.146, 13.316]
  MoveL 3556 to (238.22, 42.15, 59.84) mm, rotated rx -180 ry 0 rz 180 deg; joints [-28.315, 48.939, -75.459, 31.054, 113.146, 13.316]
  Call Extruder(206.22057)
  MoveL 3557 to (238.4, 42.45, 59.84) mm, rotated rx -180 ry 0 rz 180 deg; joints [-28.434, 48.969, -75.457, 31.172, 113.092, 13.348]
  MoveL 3558 to (238.4, 42.45, 59.84) mm, rotated rx -180 ry 0 rz 180 deg; joints [-28.434, 48.969, -75.457, 31.172, 113.092, 13.348]
  Call Extruder(206.42751)
  MoveL 3559 to (238.57, 42.75, 59.84) mm, rotated rx -180 ry 0 rz -180 deg; joints [-28.552, 48.999, -75.455, 31.29, 113.038, 13.379]
  MoveL 3560 to (238.57, 42.75, 59.84) mm, rotated rx -180 ry 0 rz -180 deg; joints [-28.552, 48.999, -75.455, 31.29, 113.038, 13.379]
  Call Extruder(206.63368)
  MoveL 3561 to (238.75, 43.06, 59.84) mm, rotated rx -180 ry 0 rz -180 deg; joints [-28.669, 49.028, -75.454, 31.407, 112.984, 13.41]
  MoveL 3562 to (238.75, 43.06, 59.84) mm, rotated rx -180 ry 0 rz -180 deg; joints [-28.669, 49.028, -75.454, 31.407, 112.984, 13.41]
  Call Extruder(206.81537)
  MoveL 3563 to (238.89, 43.33, 59.84) mm, rotated rx -180 ry 0 rz 180 deg; joints [-28.78, 49.054, -75.452, 31.519, 112.935, 13.44]
  MoveL 3564 to (238.89, 43.33, 59.84) mm, rotated rx -180 ry 0 rz 180 deg; joints [-28.78, 49.054, -75.452, 31.519, 112.935, 13.44]
  Call Extruder(206.97338)
  MoveL 3565 to (239, 43.58, 59.84) mm, rotated rx -180 ry 0 rz 180 deg; joints [-28.886, 49.075, -75.451, 31.626, 112.892, 13.471]
  MoveL 3566 to (239, 43.58, 59.84) mm, rotated rx -180 ry 0 rz 180 deg; joints [-28.886, 49.075, -75.451, 31.626, 112.892, 13.471]
  Call Extruder(207.13078)
  MoveL 3567 to (239.1, 43.83, 59.84) mm, rotated rx -180 ry 0 rz -180 deg; joints [-28.991, 49.096, -75.45, 31.732, 112.848, 13.502]
  MoveL 3568 to (239.1, 43.83, 59.84) mm, rotated rx -180 ry 0 rz -180 deg; joints [-28.991, 49.096, -75.45, 31.732, 112.848, 13.502]
  Call Extruder(207.31350)
  MoveL 3569 to (239.22, 44.12, 59.84) mm, rotated rx -180 ry 0 rz -180 deg; joints [-29.116, 49.12, -75.448, 31.858, 112.797, 13.538]
  MoveL 3570 to (239.22, 44.12, 59.84) mm, rotated rx -180 ry 0 rz -180 deg; joints [-29.116, 49.12, -75.448, 31.858, 112.797, 13.538]
  Call Extruder(207.49546)
  MoveL 3571 to (239.35, 44.42, 59.84) mm, rotated rx 180 ry 0 rz 180 deg; joints [-29.24, 49.145, -75.447, 31.982, 112.746, 13.574]
  MoveL 3572 to (239.35, 44.42, 59.84) mm, rotated rx 180 ry 0 rz 180 deg; joints [-29.24, 49.145, -75.447, 31.982, 112.746, 13.574]
  Call Extruder(207.64279)
  MoveL 3573 to (239.44, 44.66, 59.84) mm, rotated rx 180 ry 0 rz 180 deg; joints [-29.343, 49.164, -75.446, 32.087, 112.704, 13.604]
  MoveL 3574 to (239.44, 44.66, 59.84) mm, rotated rx 180 ry 0 rz 180 deg; joints [-29.343, 49.164, -75.446, 32.087, 112.704, 13.604]
  Call Extruder(207.75602)
  MoveL 3575 to (239.5, 44.85, 59.84) mm, rotated rx -180 ry 0 rz -180 deg; joints [-29.428, 49.178, -75.445, 32.172, 112.671, 13.629]
  MoveL 3576 to (239.5, 44.85, 59.84) mm, rotated rx -180 ry 0 rz -180 deg; joints [-29.428, 49.178, -75.445, 32.172, 112.671, 13.629]
  Call Extruder(207.86881)
  MoveL 3577 to (239.56, 45.03, 59.84) mm, rotated rx -180 ry 0 rz -180 deg; joints [-29.512, 49.193, -75.444, 32.257, 112.639, 13.655]
  MoveL 3578 to (239.56, 45.03, 59.84) mm, rotated rx -180 ry 0 rz -180 deg; joints [-29.512, 49.193, -75.444, 32.257, 112.639, 13.655]
  Call Extruder(207.98116)
  MoveL 3579 to (239.62, 45.22, 59.84) mm, rotated rx -180 ry 0 rz 180 deg; joints [-29.596, 49.207, -75.443, 32.342, 112.606, 13.68]
  MoveL 3580 to (239.62, 45.22, 59.84) mm, rotated rx -180 ry 0 rz 180 deg; joints [-29.596, 49.207, -75.443, 32.342, 112.606, 13.68]
  Call Extruder(208.09306)
  MoveL 3581 to (239.68, 45.41, 59.84) mm, rotated rx 180 ry 0 rz 180 deg; joints [-29.679, 49.221, -75.442, 32.427, 112.573, 13.705]
  MoveL 3582 to (239.68, 45.41, 59.84) mm, rotated rx 180 ry 0 rz 180 deg; joints [-29.679, 49.221, -75.442, 32.427, 112.573, 13.705]
  Call Extruder(208.21446)
  MoveL 3583 to (239.75, 45.62, 59.84) mm, rotated rx -180 ry 0 rz 180 deg; joints [-29.77, 49.237, -75.441, 32.519, 112.538, 13.732]
  MoveL 3584 to (239.75, 45.62, 59.84) mm, rotated rx -180 ry 0 rz 180 deg; joints [-29.77, 49.237, -75.441, 32.519, 112.538, 13.732]
  Call Extruder(208.34525)
  MoveL 3585 to (239.82, 45.84, 59.84) mm, rotated rx 180 ry 0 rz 180 deg; joints [-29.871, 49.254, -75.44, 32.62, 112.499, 13.762]
  MoveL 3586 to (239.82, 45.84, 59.84) mm, rotated rx 180 ry 0 rz 180 deg; joints [-29.871, 49.254, -75.44, 32.62, 112.499, 13.762]
  Call Extruder(208.47548)
  MoveL 3587 to (239.88, 46.06, 59.84) mm, rotated rx 180 ry 0 rz 180 deg; joints [-29.97, 49.27, -75.439, 32.721, 112.46, 13.791]
  MoveL 3588 to (239.88, 46.06, 59.84) mm, rotated rx 180 ry 0 rz 180 deg; joints [-29.97, 49.27, -75.439, 32.721, 112.46, 13.791]
  Call Extruder(208.60514)
  MoveL 3589 to (239.95, 46.29, 59.84) mm, rotated rx -180 ry 0 rz 180 deg; joints [-30.069, 49.287, -75.438, 32.821, 112.421, 13.821]
  MoveL 3590 to (239.95, 46.29, 59.84) mm, rotated rx -180 ry 0 rz 180 deg; joints [-30.069, 49.287, -75.438, 32.821, 112.421, 13.821]
  Call Extruder(208.73424)
  MoveL 3591 to (240.02, 46.51, 59.84) mm, rotated rx -180 ry 0 rz -180 deg; joints [-30.168, 49.304, -75.437, 32.922, 112.383, 13.85]
  MoveL 3592 to (240.02, 46.51, 59.84) mm, rotated rx -180 ry 0 rz -180 deg; joints [-30.168, 49.304, -75.437, 32.922, 112.383, 13.85]
  Call Extruder(208.84929)
  MoveL 3593 to (240.06, 46.72, 59.84) mm, rotated rx 180 ry 0 rz 180 deg; joints [-30.263, 49.318, -75.436, 33.018, 112.348, 13.879]
  MoveL 3594 to (240.06, 46.72, 59.84) mm, rotated rx 180 ry 0 rz 180 deg; joints [-30.263, 49.318, -75.436, 33.018, 112.348, 13.879]
  Call Extruder(208.96389)
  MoveL 3595 to (240.11, 46.92, 59.84) mm, rotated rx -180 ry 0 rz 180 deg; joints [-30.358, 49.332, -75.435, 33.114, 112.312, 13.908]
  MoveL 3596 to (240.11, 46.92, 59.84) mm, rotated rx -180 ry 0 rz 180 deg; joints [-30.358, 49.332, -75.435, 33.114, 112.312, 13.908]
  Call Extruder(209.07804)
  MoveL 3597 to (240.15, 47.12, 59.84) mm, rotated rx 180 ry 0 rz 180 deg; joints [-30.453, 49.346, -75.434, 33.21, 112.277, 13.937]
  MoveL 3598 to (240.15, 47.12, 59.84) mm, rotated rx 180 ry 0 rz 180 deg; joints [-30.453, 49.346, -75.434, 33.21, 112.277, 13.937]
  Call Extruder(209.19174)
  MoveL 3599 to (240.2, 47.33, 59.84) mm, rotated rx -180 ry 0 rz 180 deg; joints [-30.548, 49.36, -75.433, 33.306, 112.242, 13.966]
  MoveL 3600 to (240.2, 47.33, 59.84) mm, rotated rx -180 ry 0 rz 180 deg; joints [-30.548, 49.36, -75.433, 33.306, 112.242, 13.966]
  Call Extruder(209.31715)
  MoveL 3601 to (240.24, 47.56, 59.84) mm, rotated rx -180 ry 0 rz 180 deg; joints [-30.653, 49.375, -75.432, 33.412, 112.203, 13.998]
  MoveL 3602 to (240.24, 47.56, 59.84) mm, rotated rx -180 ry 0 rz 180 deg; joints [-30.653, 49.375, -75.432, 33.412, 112.203, 13.998]
  Call Extruder(209.45413)
  MoveL 3603 to (240.29, 47.8, 59.84) mm, rotated rx 180 ry 0 rz 180 deg; joints [-30.768, 49.391, -75.43, 33.53, 112.16, 14.033]
  MoveL 3604 to (240.29, 47.8, 59.84) mm, rotated rx 180 ry 0 rz 180 deg; joints [-30.768, 49.391, -75.43, 33.53, 112.16, 14.033]
  Call Extruder(209.59050)
  MoveL 3605 to (240.34, 48.05, 59.84) mm, rotated rx 180 ry 0 rz 180 deg; joints [-30.884, 49.408, -75.429, 33.647, 112.117, 14.068]
  MoveL 3606 to (240.34, 48.05, 59.84) mm, rotated rx 180 ry 0 rz 180 deg; joints [-30.884, 49.408, -75.429, 33.647, 112.117, 14.068]
  Call Extruder(209.72625)
  MoveL 3607 to (240.39, 48.3, 59.84) mm, rotated rx -180 ry 0 rz 180 deg; joints [-30.999, 49.425, -75.428, 33.763, 112.074, 14.103]
  MoveL 3608 to (240.39, 48.3, 59.84) mm, rotated rx -180 ry 0 rz 180 deg; joints [-30.999, 49.425, -75.428, 33.763, 112.074, 14.103]
  Call Extruder(209.86140)
  MoveL 3609 to (240.44, 48.55, 59.84) mm, rotated rx -180 ry 0 rz 180 deg; joints [-31.114, 49.442, -75.427, 33.879, 112.031, 14.137]
  MoveL 3610 to (240.44, 48.55, 59.84) mm, rotated rx -180 ry 0 rz 180 deg; joints [-31.114, 49.442, -75.427, 33.879, 112.031, 14.137]
  Call Extruder(209.99594)
  MoveL 3611 to (240.49, 48.8, 59.84) mm, rotated rx -180 ry 0 rz 180 deg; joints [-31.228, 49.458, -75.426, 33.995, 111.988, 14.171]
  MoveL 3612 to (240.49, 48.8, 59.84) mm, rotated rx -180 ry 0 rz 180 deg; joints [-31.228, 49.458, -75.426, 33.995, 111.988, 14.171]
  Call Extruder(210.12986)
  MoveL 3613 to (240.54, 49.05, 59.84) mm, rotated rx 180 ry 0 rz 180 deg; joints [-31.342, 49.475, -75.424, 34.11, 111.945, 14.204]
  MoveL 3614 to (240.54, 49.05, 59.84) mm, rotated rx 180 ry 0 rz 180 deg; joints [-31.342, 49.475, -75.424, 34.11, 111.945, 14.204]
  Call Extruder(210.27773)
  MoveL 3615 to (240.59, 49.33, 59.84) mm, rotated rx -180 ry 0 rz 180 deg; joints [-31.47, 49.493, -75.423, 34.239, 111.898, 14.243]
  MoveL 3616 to (240.59, 49.33, 59.84) mm, rotated rx -180 ry 0 rz 180 deg; joints [-31.47, 49.493, -75.423, 34.239, 111.898, 14.243]
  Call Extruder(210.43947)
  MoveL 3617 to (240.64, 49.63, 59.84) mm, rotated rx -180 ry 0 rz 180 deg; joints [-31.612, 49.513, -75.422, 34.383, 111.845, 14.285]
  MoveL 3618 to (240.64, 49.63, 59.84) mm, rotated rx -180 ry 0 rz 180 deg; joints [-31.612, 49.513, -75.422, 34.383, 111.845, 14.285]
  Call Extruder(210.60049)
  MoveL 3619 to (240.69, 49.94, 59.84) mm, rotated rx 180 ry 0 rz 180 deg; joints [-31.755, 49.533, -75.42, 34.527, 111.793, 14.327]
  MoveL 3620 to (240.69, 49.94, 59.84) mm, rotated rx 180 ry 0 rz 180 deg; joints [-31.755, 49.533, -75.42, 34.527, 111.793, 14.327]
  Call Extruder(210.76078)
  MoveL 3621 to (240.74, 50.24, 59.84) mm, rotated rx -180 ry 0 rz 180 deg; joints [-31.895, 49.552, -75.418, 34.669, 111.74, 14.369]
  MoveL 3622 to (240.74, 50.24, 59.84) mm, rotated rx -180 ry 0 rz 180 deg; joints [-31.895, 49.552, -75.418, 34.669, 111.74, 14.369]
  Call Extruder(210.92034)
  MoveL 3623 to (240.78, 50.55, 59.84) mm, rotated rx -180 ry 0 rz 180 deg; joints [-32.036, 49.572, -75.417, 34.811, 111.688, 14.41]
  MoveL 3624 to (240.78, 50.55, 59.84) mm, rotated rx -180 ry 0 rz 180 deg; joints [-32.036, 49.572, -75.417, 34.811, 111.688, 14.41]
  Call Extruder(211.07917)
  MoveL 3625 to (240.83, 50.86, 59.84) mm, rotated rx 180 ry 0 rz 180 deg; joints [-32.176, 49.592, -75.415, 34.952, 111.635, 14.451]
  MoveL 3626 to (240.83, 50.86, 59.84) mm, rotated rx 180 ry 0 rz 180 deg; joints [-32.176, 49.592, -75.415, 34.952, 111.635, 14.451]
  Call Extruder(211.25784)
  MoveL 3627 to (240.88, 51.2, 59.84) mm, rotated rx -180 ry 0 rz 180 deg; joints [-32.337, 49.614, -75.414, 35.113, 111.576, 14.498]
  MoveL 3628 to (240.88, 51.2, 59.84) mm, rotated rx -180 ry 0 rz 180 deg; joints [-32.337, 49.614, -75.414, 35.113, 111.576, 14.498]
  Call Extruder(211.45628)
  MoveL 3629 to (240.93, 51.59, 59.84) mm, rotated rx 180 ry 0 rz 180 deg; joints [-32.518, 49.638, -75.412, 35.296, 111.509, 14.551]
  MoveL 3630 to (240.93, 51.59, 59.84) mm, rotated rx 180 ry 0 rz 180 deg; joints [-32.518, 49.638, -75.412, 35.296, 111.509, 14.551]
  Call Extruder(211.65386)
  MoveL 3631 to (240.97, 51.98, 59.84) mm, rotated rx -180 ry 0 rz 180 deg; joints [-32.697, 49.662, -75.41, 35.477, 111.443, 14.603]
  MoveL 3632 to (240.97, 51.98, 59.84) mm, rotated rx -180 ry 0 rz 180 deg; joints [-32.697, 49.662, -75.41, 35.477, 111.443, 14.603]
  Call Extruder(211.85056)
  MoveL 3633 to (241.02, 52.36, 59.84) mm, rotated rx 180 ry 0 rz 180 deg; joints [-32.876, 49.686, -75.408, 35.657, 111.376, 14.654]
  MoveL 3634 to (241.02, 52.36, 59.84) mm, rotated rx 180 ry 0 rz 180 deg; joints [-32.876, 49.686, -75.408, 35.657, 111.376, 14.654]
  Call Extruder(212.04640)
  MoveL 3635 to (241.06, 52.75, 59.84) mm, rotated rx 180 ry 0 rz -180 deg; joints [-33.055, 49.71, -75.406, 35.836, 111.31, 14.705]
  MoveL 3636 to (241.06, 52.75, 59.84) mm, rotated rx 180 ry 0 rz -180 deg; joints [-33.055, 49.71, -75.406, 35.836, 111.31, 14.705]
  Call Extruder(212.34184)
  MoveL 3637 to (241.11, 53.34, 59.84) mm, rotated rx -180 ry 0 rz 180 deg; joints [-33.331, 49.746, -75.403, 36.114, 111.208, 14.785]
  MoveL 3638 to (241.11, 53.34, 59.84) mm, rotated rx -180 ry 0 rz 180 deg; joints [-33.331, 49.746, -75.403, 36.114, 111.208, 14.785]
  Call Extruder(212.63595)
  MoveL 3639 to (241.16, 53.93, 59.84) mm, rotated rx 180 ry 0 rz 180 deg; joints [-33.606, 49.781, -75.4, 36.39, 111.107, 14.864]
  MoveL 3640 to (241.16, 53.93, 59.84) mm, rotated rx 180 ry 0 rz 180 deg; joints [-33.606, 49.781, -75.4, 36.39, 111.107, 14.864]
  Call Extruder(212.92873)
  MoveL 3641 to (241.2, 54.52, 59.84) mm, rotated rx -180 ry 0 rz 180 deg; joints [-33.878, 49.816, -75.396, 36.664, 111.006, 14.941]
  MoveL 3642 to (241.2, 54.52, 59.84) mm, rotated rx -180 ry 0 rz 180 deg; joints [-33.878, 49.816, -75.396, 36.664, 111.006, 14.941]
  Call Extruder(213.50218)
  MoveL 3643 to (241.25, 55.68, 59.84) mm, rotated rx 180 ry 0 rz 180 deg; joints [-34.425, 49.883, -75.39, 37.212, 110.806, 15.095]
  MoveL 3644 to (241.25, 55.68, 59.84) mm, rotated rx 180 ry 0 rz 180 deg; joints [-34.425, 49.883, -75.39, 37.212, 110.806, 15.095]
  Call Extruder(214.21601)
  MoveL 3645 to (241.29, 57.14, 59.84) mm, rotated rx -180 ry 0 rz 180 deg; joints [-35.104, 49.967, -75.383, 37.891, 110.556, 15.283]
  Call Extruder(256.28089)
  MoveL 3646 to (241.29, 142.86, 59.84) mm, rotated rx 180 ry 0 rz 180 deg; joints [-60.361, 55.735, -73.982, 61.614, 98.908, 15.99]
  Call Extruder(256.70932)
  MoveL 3647 to (241.27, 143.73, 59.84) mm, rotated rx -180 ry 0 rz 180 deg; joints [-60.516, 55.796, -73.957, 61.753, 98.824, 15.936]
  MoveL 3648 to (241.27, 143.73, 59.84) mm, rotated rx -180 ry 0 rz 180 deg; joints [-60.516, 55.796, -73.957, 61.753, 98.824, 15.936]
  Call Extruder(257.28277)
  MoveL 3649 to (241.22, 144.9, 59.84) mm, rotated rx 180 ry 0 rz 180 deg; joints [-60.726, 55.875, -73.923, 61.943, 98.713, 15.866]
  MoveL 3650 to (241.22, 144.9, 59.84) mm, rotated rx 180 ry 0 rz 180 deg; joints [-60.726, 55.875, -73.923, 61.943, 98.713, 15.866]
  Call Extruder(257.71711)
  MoveL 3651 to (241.18, 145.77, 59.84) mm, rotated rx 180 ry 0 rz 180 deg; joints [-60.887, 55.935, -73.897, 62.088, 98.629, 15.814]
  MoveL 3652 to (241.18, 145.77, 59.84) mm, rotated rx 180 ry 0 rz 180 deg; joints [-60.887, 55.935, -73.897, 62.088, 98.629, 15.814]
  Call Extruder(258.01122)
  MoveL 3653 to (241.13, 146.36, 59.84) mm, rotated rx 180 ry 0 rz 180 deg; joints [-61, 55.974, -73.88, 62.19, 98.572, 15.78]
  MoveL 3654 to (241.13, 146.36, 59.84) mm, rotated rx 180 ry 0 rz 180 deg; joints [-61, 55.974, -73.88, 62.19, 98.572, 15.78]
  Call Extruder(258.30666)
  MoveL 3655 to (241.09, 146.95, 59.84) mm, rotated rx 180 ry 0 rz 180 deg; joints [-61.111, 56.013, -73.862, 62.291, 98.516, 15.745]
  MoveL 3656 to (241.09, 146.95, 59.84) mm, rotated rx 180 ry 0 rz 180 deg; joints [-61.111, 56.013, -73.862, 62.291, 98.516, 15.745]
  Call Extruder(258.55291)
  MoveL 3657 to (241.04, 147.44, 59.84) mm, rotated rx 180 ry 0 rz 180 deg; joints [-61.205, 56.045, -73.848, 62.376, 98.469, 15.717]
  MoveL 3658 to (241.04, 147.44, 59.84) mm, rotated rx 180 ry 0 rz 180 deg; joints [-61.205, 56.045, -73.848, 62.376, 98.469, 15.717]
  Call Extruder(258.74962)
  MoveL 3659 to (240.99, 147.83, 59.84) mm, rotated rx 180 ry 0 rz 180 deg; joints [-61.282, 56.071, -73.837, 62.446, 98.431, 15.695]
  MoveL 3660 to (240.99, 147.83, 59.84) mm, rotated rx 180 ry 0 rz 180 deg; joints [-61.282, 56.071, -73.837, 62.446, 98.431, 15.695]
  Call Extruder(258.94719)
  MoveL 3661 to (240.95, 148.22, 59.84) mm, rotated rx -180 ry 0 rz 180 deg; joints [-61.359, 56.096, -73.825, 62.516, 98.393, 15.674]
  MoveL 3662 to (240.95, 148.22, 59.84) mm, rotated rx -180 ry 0 rz 180 deg; joints [-61.359, 56.096, -73.825, 62.516, 98.393, 15.674]
  Call Extruder(259.14563)
  MoveL 3663 to (240.9, 148.6, 59.84) mm, rotated rx 180 ry 0 rz -180 deg; joints [-61.436, 56.121, -73.814, 62.586, 98.356, 15.652]
  MoveL 3664 to (240.9, 148.6, 59.84) mm, rotated rx 180 ry 0 rz -180 deg; joints [-61.436, 56.121, -73.814, 62.586, 98.356, 15.652]
  Call Extruder(259.34494)
  MoveL 3665 to (240.86, 148.99, 59.84) mm, rotated rx 180 ry 0 rz 180 deg; joints [-61.512, 56.146, -73.803, 62.655, 98.318, 15.63]
  MoveL 3666 to (240.86, 148.99, 59.84) mm, rotated rx 180 ry 0 rz 180 deg; joints [-61.512, 56.146, -73.803, 62.655, 98.318, 15.63]
  Call Extruder(259.50377)
  MoveL 3667 to (240.81, 149.3, 59.84) mm, rotated rx 180 ry 0 rz 180 deg; joints [-61.575, 56.166, -73.794, 62.714, 98.288, 15.613]
  MoveL 3668 to (240.81, 149.3, 59.84) mm, rotated rx 180 ry 0 rz 180 deg; joints [-61.575, 56.166, -73.794, 62.714, 98.288, 15.613]
  Call Extruder(259.66333)
  MoveL 3669 to (240.76, 149.6, 59.84) mm, rotated rx -180 ry 0 rz 180 deg; joints [-61.639, 56.185, -73.785, 62.772, 98.258, 15.597]
  MoveL 3670 to (240.76, 149.6, 59.84) mm, rotated rx -180 ry 0 rz 180 deg; joints [-61.639, 56.185, -73.785, 62.772, 98.258, 15.597]
  Call Extruder(259.82362)
  MoveL 3671 to (240.71, 149.91, 59.84) mm, rotated rx 180 ry 0 rz 180 deg; joints [-61.702, 56.204, -73.776, 62.829, 98.228, 15.58]
  MoveL 3672 to (240.71, 149.91, 59.84) mm, rotated rx 180 ry 0 rz 180 deg; joints [-61.702, 56.204, -73.776, 62.829, 98.228, 15.58]
  Call Extruder(259.98464)
  MoveL 3673 to (240.66, 150.21, 59.84) mm, rotated rx -180 ry 0 rz -180 deg; joints [-61.765, 56.224, -73.767, 62.887, 98.198, 15.563]
  MoveL 3674 to (240.66, 150.21, 59.84) mm, rotated rx -180 ry 0 rz -180 deg; joints [-61.765, 56.224, -73.767, 62.887, 98.198, 15.563]
  Call Extruder(260.14638)
  MoveL 3675 to (240.61, 150.52, 59.84) mm, rotated rx 180 ry 0 rz -180 deg; joints [-61.828, 56.243, -73.758, 62.945, 98.169, 15.547]
  MoveL 3676 to (240.61, 150.52, 59.84) mm, rotated rx 180 ry 0 rz -180 deg; joints [-61.828, 56.243, -73.758, 62.945, 98.169, 15.547]
  Call Extruder(260.30885)
  MoveL 3677 to (240.56, 150.83, 59.84) mm, rotated rx -180 ry 0 rz 180 deg; joints [-61.891, 56.263, -73.749, 63.002, 98.139, 15.53]
  MoveL 3678 to (240.56, 150.83, 59.84) mm, rotated rx -180 ry 0 rz 180 deg; joints [-61.891, 56.263, -73.749, 63.002, 98.139, 15.53]
  Call Extruder(260.44278)
  MoveL 3679 to (240.52, 151.07, 59.84) mm, rotated rx -180 ry 0 rz 180 deg; joints [-61.944, 56.278, -73.742, 63.052, 98.114, 15.517]
  MoveL 3680 to (240.52, 151.07, 59.84) mm, rotated rx -180 ry 0 rz 180 deg; joints [-61.944, 56.278, -73.742, 63.052, 98.114, 15.517]
  Call Extruder(260.57732)
  MoveL 3681 to (240.47, 151.32, 59.84) mm, rotated rx -180 ry 0 rz 180 deg; joints [-61.998, 56.294, -73.735, 63.101, 98.09, 15.504]
  MoveL 3682 to (240.47, 151.32, 59.84) mm, rotated rx -180 ry 0 rz 180 deg; joints [-61.998, 56.294, -73.735, 63.101, 98.09, 15.504]
  Call Extruder(260.71246)
  MoveL 3683 to (240.42, 151.57, 59.84) mm, rotated rx -180 ry 0 rz 180 deg; joints [-62.052, 56.309, -73.728, 63.151, 98.065, 15.491]
  MoveL 3684 to (240.42, 151.57, 59.84) mm, rotated rx -180 ry 0 rz 180 deg; joints [-62.052, 56.309, -73.728, 63.151, 98.065, 15.491]
  Call Extruder(260.84822)
  MoveL 3685 to (240.37, 151.82, 59.84) mm, rotated rx -180 ry 0 rz 180 deg; joints [-62.105, 56.325, -73.721, 63.2, 98.041, 15.478]
  MoveL 3686 to (240.37, 151.82, 59.84) mm, rotated rx -180 ry 0 rz 180 deg; joints [-62.105, 56.325, -73.721, 63.2, 98.041, 15.478]
  Call Extruder(260.98459)
  MoveL 3687 to (240.32, 152.07, 59.84) mm, rotated rx 180 ry 0 rz 180 deg; joints [-62.159, 56.34, -73.713, 63.249, 98.016, 15.464]
  MoveL 3688 to (240.32, 152.07, 59.84) mm, rotated rx 180 ry 0 rz 180 deg; joints [-62.159, 56.34, -73.713, 63.249, 98.016, 15.464]
  Call Extruder(261.12157)
  MoveL 3689 to (240.27, 152.32, 59.84) mm, rotated rx 180 ry 0 rz -180 deg; joints [-62.212, 56.355, -73.706, 63.298, 97.992, 15.451]
  MoveL 3690 to (240.27, 152.32, 59.84) mm, rotated rx 180 ry 0 rz -180 deg; joints [-62.212, 56.355, -73.706, 63.298, 97.992, 15.451]
  Call Extruder(261.25915)
  MoveL 3691 to (240.22, 152.57, 59.84) mm, rotated rx 180 ry 0 rz 180 deg; joints [-62.265, 56.371, -73.699, 63.347, 97.967, 15.438]
  MoveL 3692 to (240.22, 152.57, 59.84) mm, rotated rx 180 ry 0 rz 180 deg; joints [-62.265, 56.371, -73.699, 63.347, 97.967, 15.438]
  Call Extruder(261.37285)
  MoveL 3693 to (240.17, 152.77, 59.84) mm, rotated rx -180 ry 0 rz 180 deg; joints [-62.31, 56.383, -73.693, 63.388, 97.947, 15.427]
  MoveL 3694 to (240.17, 152.77, 59.84) mm, rotated rx -180 ry 0 rz 180 deg; joints [-62.31, 56.383, -73.693, 63.388, 97.947, 15.427]
  Call Extruder(261.48700)
  MoveL 3695 to (240.13, 152.98, 59.84) mm, rotated rx -180 ry 0 rz 180 deg; joints [-62.355, 56.396, -73.687, 63.429, 97.927, 15.416]
  MoveL 3696 to (240.13, 152.98, 59.84) mm, rotated rx -180 ry 0 rz 180 deg; joints [-62.355, 56.396, -73.687, 63.429, 97.927, 15.416]
  Call Extruder(261.60161)
  MoveL 3697 to (240.08, 153.18, 59.84) mm, rotated rx -180 ry 0 rz 180 deg; joints [-62.399, 56.408, -73.681, 63.47, 97.907, 15.406]
  MoveL 3698 to (240.08, 153.18, 59.84) mm, rotated rx -180 ry 0 rz 180 deg; joints [-62.399, 56.408, -73.681, 63.47, 97.907, 15.406]
  Call Extruder(261.71666)
  MoveL 3699 to (240.04, 153.39, 59.84) mm, rotated rx -180 ry 0 rz -180 deg; joints [-62.444, 56.421, -73.675, 63.511, 97.887, 15.395]
  MoveL 3700 to (240.04, 153.39, 59.84) mm, rotated rx -180 ry 0 rz -180 deg; joints [-62.444, 56.421, -73.675, 63.511, 97.887, 15.395]
  Call Extruder(261.83888)
  MoveL 3701 to (239.98, 153.6, 59.84) mm, rotated rx 180 ry 0 rz 180 deg; joints [-62.493, 56.434, -73.669, 63.557, 97.865, 15.384]
  MoveL 3702 to (239.98, 153.6, 59.84) mm, rotated rx 180 ry 0 rz 180 deg; joints [-62.493, 56.434, -73.669, 63.557, 97.865, 15.384]
  Call Extruder(261.96855)
  MoveL 3703 to (239.92, 153.82, 59.84) mm, rotated rx 180 ry 0 rz -180 deg; joints [-62.547, 56.447, -73.663, 63.607, 97.843, 15.374]
  MoveL 3704 to (239.92, 153.82, 59.84) mm, rotated rx 180 ry 0 rz -180 deg; joints [-62.547, 56.447, -73.663, 63.607, 97.843, 15.374]
  Call Extruder(262.09877)
  MoveL 3705 to (239.85, 154.05, 59.84) mm, rotated rx -180 ry 0 rz 180 deg; joints [-62.601, 56.46, -73.657, 63.657, 97.82, 15.364]
  MoveL 3706 to (239.85, 154.05, 59.84) mm, rotated rx -180 ry 0 rz 180 deg; joints [-62.601, 56.46, -73.657, 63.657, 97.82, 15.364]
  Call Extruder(262.22956)
  MoveL 3707 to (239.78, 154.27, 59.84) mm, rotated rx 180 ry 0 rz 180 deg; joints [-62.654, 56.473, -73.65, 63.707, 97.797, 15.354]
  MoveL 3708 to (239.78, 154.27, 59.84) mm, rotated rx 180 ry 0 rz 180 deg; joints [-62.654, 56.473, -73.65, 63.707, 97.797, 15.354]
  Call Extruder(262.36092)
  MoveL 3709 to (239.71, 154.49, 59.84) mm, rotated rx -180 ry 0 rz 180 deg; joints [-62.708, 56.486, -73.644, 63.757, 97.774, 15.343]
  MoveL 3710 to (239.71, 154.49, 59.84) mm, rotated rx -180 ry 0 rz 180 deg; joints [-62.708, 56.486, -73.644, 63.757, 97.774, 15.343]
  Call Extruder(262.47282)
  MoveL 3711 to (239.65, 154.68, 59.84) mm, rotated rx -180 ry 0 rz 180 deg; joints [-62.754, 56.497, -73.639, 63.8, 97.755, 15.335]
  MoveL 3712 to (239.65, 154.68, 59.84) mm, rotated rx -180 ry 0 rz 180 deg; joints [-62.754, 56.497, -73.639, 63.8, 97.755, 15.335]
  Call Extruder(262.58516)
  MoveL 3713 to (239.59, 154.87, 59.84) mm, rotated rx -180 ry 0 rz 180 deg; joints [-62.801, 56.508, -73.634, 63.843, 97.735, 15.326]
  MoveL 3714 to (239.59, 154.87, 59.84) mm, rotated rx -180 ry 0 rz 180 deg; joints [-62.801, 56.508, -73.634, 63.843, 97.735, 15.326]
  Call Extruder(262.69795)
  MoveL 3715 to (239.53, 155.06, 59.84) mm, rotated rx -180 ry 0 rz 180 deg; joints [-62.847, 56.519, -73.628, 63.886, 97.716, 15.318]
  MoveL 3716 to (239.53, 155.06, 59.84) mm, rotated rx -180 ry 0 rz 180 deg; joints [-62.847, 56.519, -73.628, 63.886, 97.716, 15.318]
  Call Extruder(262.81119)
  MoveL 3717 to (239.47, 155.25, 59.84) mm, rotated rx -180 ry 0 rz 180 deg; joints [-62.893, 56.53, -73.623, 63.929, 97.697, 15.309]
  MoveL 3718 to (239.47, 155.25, 59.84) mm, rotated rx -180 ry 0 rz 180 deg; joints [-62.893, 56.53, -73.623, 63.929, 97.697, 15.309]
  Call Extruder(262.92487)
  MoveL 3719 to (239.41, 155.44, 59.84) mm, rotated rx 180 ry 0 rz 180 deg; joints [-62.939, 56.54, -73.618, 63.972, 97.678, 15.3]
  MoveL 3720 to (239.41, 155.44, 59.84) mm, rotated rx 180 ry 0 rz 180 deg; joints [-62.939, 56.54, -73.618, 63.972, 97.678, 15.3]
  Call Extruder(263.10683)
  MoveL 3721 to (239.29, 155.73, 59.84) mm, rotated rx 180 ry 0 rz 180 deg; joints [-63.018, 56.556, -73.61, 64.046, 97.646, 15.289]
  MoveL 3722 to (239.29, 155.73, 59.84) mm, rotated rx 180 ry 0 rz 180 deg; joints [-63.018, 56.556, -73.61, 64.046, 97.646, 15.289]
  Call Extruder(263.28954)
  MoveL 3723 to (239.16, 156.02, 59.84) mm, rotated rx -180 ry 0 rz 180 deg; joints [-63.097, 56.572, -73.602, 64.12, 97.615, 15.278]
  MoveL 3724 to (239.16, 156.02, 59.84) mm, rotated rx -180 ry 0 rz 180 deg; joints [-63.097, 56.572, -73.602, 64.12, 97.615, 15.278]
  Call Extruder(263.45997)
  MoveL 3725 to (239.05, 156.29, 59.84) mm, rotated rx 180 ry 0 rz -180 deg; joints [-63.17, 56.587, -73.595, 64.188, 97.586, 15.267]
  MoveL 3726 to (239.05, 156.29, 59.84) mm, rotated rx 180 ry 0 rz -180 deg; joints [-63.17, 56.587, -73.595, 64.188, 97.586, 15.267]
  Call Extruder(263.61798)
  MoveL 3727 to (238.94, 156.54, 59.84) mm, rotated rx -180 ry 0 rz 180 deg; joints [-63.238, 56.6, -73.588, 64.252, 97.56, 15.258]
  MoveL 3728 to (238.94, 156.54, 59.84) mm, rotated rx -180 ry 0 rz 180 deg; joints [-63.238, 56.6, -73.588, 64.252, 97.56, 15.258]
  Call Extruder(263.77659)
  MoveL 3729 to (238.84, 156.79, 59.84) mm, rotated rx -180 ry 0 rz -180 deg; joints [-63.306, 56.614, -73.582, 64.316, 97.533, 15.248]
  MoveL 3730 to (238.84, 156.79, 59.84) mm, rotated rx -180 ry 0 rz -180 deg; joints [-63.306, 56.614, -73.582, 64.316, 97.533, 15.248]
  Call Extruder(263.98276)
  MoveL 3731 to (238.66, 157.09, 59.84) mm, rotated rx -180 ry 0 rz -180 deg; joints [-63.401, 56.629, -73.574, 64.406, 97.498, 15.24]
  MoveL 3732 to (238.66, 157.09, 59.84) mm, rotated rx -180 ry 0 rz -180 deg; joints [-63.401, 56.629, -73.574, 64.406, 97.498, 15.24]
  Call Extruder(264.18971)
  MoveL 3733 to (238.49, 157.4, 59.84) mm, rotated rx -180 ry 0 rz 180 deg; joints [-63.497, 56.644, -73.567, 64.496, 97.464, 15.232]
  MoveL 3734 to (238.49, 157.4, 59.84) mm, rotated rx -180 ry 0 rz 180 deg; joints [-63.497, 56.644, -73.567, 64.496, 97.464, 15.232]
  Call Extruder(264.39743)
  MoveL 3735 to (238.31, 157.7, 59.84) mm, rotated rx 180 ry 0 rz 180 deg; joints [-63.592, 56.659, -73.56, 64.586, 97.429, 15.223]
  MoveL 3736 to (238.31, 157.7, 59.84) mm, rotated rx 180 ry 0 rz 180 deg; joints [-63.592, 56.659, -73.56, 64.586, 97.429, 15.223]
  Call Extruder(264.60594)
  MoveL 3737 to (238.13, 158.01, 59.84) mm, rotated rx -180 ry 0 rz 180 deg; joints [-63.687, 56.674, -73.552, 64.676, 97.394, 15.215]
  MoveL 3738 to (238.13, 158.01, 59.84) mm, rotated rx -180 ry 0 rz 180 deg; joints [-63.687, 56.674, -73.552, 64.676, 97.394, 15.215]
  Call Extruder(264.78548)
  MoveL 3739 to (237.96, 158.25, 59.84) mm, rotated rx 180 ry 0 rz 180 deg; joints [-63.774, 56.685, -73.547, 64.758, 97.365, 15.211]
  MoveL 3740 to (237.96, 158.25, 59.84) mm, rotated rx 180 ry 0 rz 180 deg; joints [-63.774, 56.685, -73.547, 64.758, 97.365, 15.211]
  Call Extruder(265.11889)
  MoveL 3741 to (237.63, 158.7, 59.84) mm, rotated rx 180 ry 0 rz -180 deg; joints [-63.934, 56.705, -73.537, 64.911, 97.31, 15.203]
  MoveL 3742 to (237.63, 158.7, 59.84) mm, rotated rx 180 ry 0 rz -180 deg; joints [-63.934, 56.705, -73.537, 64.911, 97.31, 15.203]
  Call Extruder(265.45348)
  MoveL 3743 to (237.3, 159.15, 59.84) mm, rotated rx -180 ry 0 rz 180 deg; joints [-64.094, 56.725, -73.526, 65.063, 97.255, 15.195]
  Call Extruder(266.28143)
  MoveL 3744 to (236.39, 160.19, 59.84) mm, rotated rx -180 ry 0 rz 180 deg; joints [-64.505, 56.767, -73.506, 65.455, 97.121, 15.188]
  Call Extruder(267.10937)
  MoveL 3745 to (235.35, 161.1, 59.84) mm, rotated rx -180 ry 0 rz -180 deg; joints [-64.933, 56.796, -73.491, 65.867, 96.991, 15.198]
  Call Extruder(267.27668)
  MoveL 3746 to (235.13, 161.27, 59.84) mm, rotated rx -180 ry 0 rz -180 deg; joints [-65.021, 56.8, -73.489, 65.952, 96.965, 15.203]
  MoveL 3747 to (235.13, 161.27, 59.84) mm, rotated rx -180 ry 0 rz -180 deg; joints [-65.021, 56.8, -73.489, 65.952, 96.965, 15.203]
  Call Extruder(267.61010)
  MoveL 3748 to (234.68, 161.59, 59.84) mm, rotated rx 180 ry 0 rz 180 deg; joints [-65.197, 56.809, -73.484, 66.122, 96.914, 15.212]
  MoveL 3749 to (234.68, 161.59, 59.84) mm, rotated rx 180 ry 0 rz 180 deg; joints [-65.197, 56.809, -73.484, 66.122, 96.914, 15.212]
  Call Extruder(267.94234)
  MoveL 3750 to (234.22, 161.92, 59.84) mm, rotated rx 180 ry 0 rz 180 deg; joints [-65.374, 56.817, -73.48, 66.292, 96.862, 15.221]
  MoveL 3751 to (234.22, 161.92, 59.84) mm, rotated rx 180 ry 0 rz 180 deg; joints [-65.374, 56.817, -73.48, 66.292, 96.862, 15.221]
  Call Extruder(268.06000)
  MoveL 3752 to (234.05, 162.02, 59.84) mm, rotated rx 180 ry 0 rz 180 deg; joints [-65.437, 56.818, -73.479, 66.353, 96.845, 15.226]
  MoveL 3753 to (234.05, 162.02, 59.84) mm, rotated rx 180 ry 0 rz 180 deg; joints [-65.437, 56.818, -73.479, 66.353, 96.845, 15.226]
  Call Extruder(268.26773)
  MoveL 3754 to (233.75, 162.2, 59.84) mm, rotated rx -180 ry 0 rz 180 deg; joints [-65.549, 56.821, -73.478, 66.462, 96.814, 15.236]
  MoveL 3755 to (233.75, 162.2, 59.84) mm, rotated rx -180 ry 0 rz 180 deg; joints [-65.549, 56.821, -73.478, 66.462, 96.814, 15.236]
  Call Extruder(268.47467)
  MoveL 3756 to (233.45, 162.37, 59.84) mm, rotated rx -180 ry 0 rz 180 deg; joints [-65.662, 56.824, -73.477, 66.57, 96.783, 15.245]
  MoveL 3757 to (233.45, 162.37, 59.84) mm, rotated rx -180 ry 0 rz 180 deg; joints [-65.662, 56.824, -73.477, 66.57, 96.783, 15.245]
  Call Extruder(268.68084)
  MoveL 3758 to (233.14, 162.55, 59.84) mm, rotated rx -180 ry 0 rz 180 deg; joints [-65.774, 56.826, -73.475, 66.679, 96.752, 15.254]
  MoveL 3759 to (233.14, 162.55, 59.84) mm, rotated rx -180 ry 0 rz 180 deg; joints [-65.774, 56.826, -73.475, 66.679, 96.752, 15.254]
  Call Extruder(268.86251)
  MoveL 3760 to (232.87, 162.69, 59.84) mm, rotated rx 180 ry 0 rz 180 deg; joints [-65.874, 56.827, -73.475, 66.776, 96.725, 15.264]
  MoveL 3761 to (232.87, 162.69, 59.84) mm, rotated rx 180 ry 0 rz 180 deg; joints [-65.874, 56.827, -73.475, 66.776, 96.725, 15.264]
  Call Extruder(269.02049)
  MoveL 3762 to (232.62, 162.8, 59.84) mm, rotated rx 180 ry 0 rz 180 deg; joints [-65.961, 56.827, -73.475, 66.86, 96.702, 15.274]
  MoveL 3763 to (232.62, 162.8, 59.84) mm, rotated rx 180 ry 0 rz 180 deg; joints [-65.961, 56.827, -73.475, 66.86, 96.702, 15.274]
  Call Extruder(269.17786)
  MoveL 3764 to (232.37, 162.9, 59.84) mm, rotated rx -180 ry 0 rz 180 deg; joints [-66.048, 56.827, -73.475, 66.945, 96.679, 15.284]
  MoveL 3765 to (232.37, 162.9, 59.84) mm, rotated rx -180 ry 0 rz 180 deg; joints [-66.048, 56.827, -73.475, 66.945, 96.679, 15.284]
  Call Extruder(269.36060)
  MoveL 3766 to (232.07, 163.03, 59.84) mm, rotated rx 180 ry 0 rz -180 deg; joints [-66.149, 56.826, -73.475, 67.044, 96.653, 15.297]
  MoveL 3767 to (232.07, 163.03, 59.84) mm, rotated rx 180 ry 0 rz -180 deg; joints [-66.149, 56.826, -73.475, 67.044, 96.653, 15.297]
  Call Extruder(269.54259)
  MoveL 3768 to (231.78, 163.15, 59.84) mm, rotated rx -180 ry 0 rz -180 deg; joints [-66.251, 56.826, -73.476, 67.142, 96.626, 15.309]
  MoveL 3769 to (231.78, 163.15, 59.84) mm, rotated rx -180 ry 0 rz -180 deg; joints [-66.251, 56.826, -73.476, 67.142, 96.626, 15.309]
  Call Extruder(269.68992)
  MoveL 3770 to (231.54, 163.24, 59.84) mm, rotated rx -180 ry 0 rz -180 deg; joints [-66.333, 56.825, -73.476, 67.223, 96.605, 15.32]
  MoveL 3771 to (231.54, 163.24, 59.84) mm, rotated rx -180 ry 0 rz -180 deg; joints [-66.333, 56.825, -73.476, 67.223, 96.605, 15.32]
  Call Extruder(269.80315)
  MoveL 3772 to (231.35, 163.3, 59.84) mm, rotated rx 180 ry 0 rz -180 deg; joints [-66.397, 56.823, -73.477, 67.285, 96.589, 15.329]
  MoveL 3773 to (231.35, 163.3, 59.84) mm, rotated rx 180 ry 0 rz -180 deg; joints [-66.397, 56.823, -73.477, 67.285, 96.589, 15.329]
  Call Extruder(269.91592)
  MoveL 3774 to (231.17, 163.36, 59.84) mm, rotated rx -180 ry 0 rz 180 deg; joints [-66.46, 56.822, -73.478, 67.346, 96.573, 15.338]
  MoveL 3775 to (231.17, 163.36, 59.84) mm, rotated rx -180 ry 0 rz 180 deg; joints [-66.46, 56.822, -73.478, 67.346, 96.573, 15.338]
  Call Extruder(270.02826)
  MoveL 3776 to (230.98, 163.42, 59.84) mm, rotated rx 180 ry 0 rz 180 deg; joints [-66.524, 56.82, -73.478, 67.408, 96.557, 15.347]
  MoveL 3777 to (230.98, 163.42, 59.84) mm, rotated rx 180 ry 0 rz 180 deg; joints [-66.524, 56.82, -73.478, 67.408, 96.557, 15.347]
  Call Extruder(270.14014)
  MoveL 3778 to (230.79, 163.48, 59.84) mm, rotated rx 180 ry 0 rz 180 deg; joints [-66.587, 56.819, -73.479, 67.47, 96.541, 15.356]
  MoveL 3779 to (230.79, 163.48, 59.84) mm, rotated rx 180 ry 0 rz 180 deg; joints [-66.587, 56.819, -73.479, 67.47, 96.541, 15.356]
  Call Extruder(270.26155)
  MoveL 3780 to (230.58, 163.55, 59.84) mm, rotated rx 180 ry 0 rz -180 deg; joints [-66.656, 56.817, -73.48, 67.537, 96.524, 15.366]
  MoveL 3781 to (230.58, 163.55, 59.84) mm, rotated rx 180 ry 0 rz -180 deg; joints [-66.656, 56.817, -73.48, 67.537, 96.524, 15.366]
  Call Extruder(270.39236)
  MoveL 3782 to (230.36, 163.61, 59.84) mm, rotated rx -180 ry 0 rz -180 deg; joints [-66.731, 56.815, -73.481, 67.61, 96.505, 15.377]
  MoveL 3783 to (230.36, 163.61, 59.84) mm, rotated rx -180 ry 0 rz -180 deg; joints [-66.731, 56.815, -73.481, 67.61, 96.505, 15.377]
  Call Extruder(270.52261)
  MoveL 3784 to (230.14, 163.68, 59.84) mm, rotated rx 180 ry 0 rz -180 deg; joints [-66.805, 56.813, -73.482, 67.683, 96.487, 15.388]
  MoveL 3785 to (230.14, 163.68, 59.84) mm, rotated rx 180 ry 0 rz -180 deg; joints [-66.805, 56.813, -73.482, 67.683, 96.487, 15.388]
  Call Extruder(270.65229)
  MoveL 3786 to (229.91, 163.75, 59.84) mm, rotated rx -180 ry 0 rz -180 deg; joints [-66.88, 56.811, -73.483, 67.756, 96.468, 15.399]
  MoveL 3787 to (229.91, 163.75, 59.84) mm, rotated rx -180 ry 0 rz -180 deg; joints [-66.88, 56.811, -73.483, 67.756, 96.468, 15.399]
  Call Extruder(270.78141)
  MoveL 3788 to (229.69, 163.82, 59.84) mm, rotated rx -180 ry 0 rz 180 deg; joints [-66.955, 56.809, -73.484, 67.828, 96.449, 15.41]
  MoveL 3789 to (229.69, 163.82, 59.84) mm, rotated rx -180 ry 0 rz 180 deg; joints [-66.955, 56.809, -73.484, 67.828, 96.449, 15.41]
  Call Extruder(270.89648)
  MoveL 3790 to (229.48, 163.86, 59.84) mm, rotated rx -180 ry 0 rz 180 deg; joints [-67.021, 56.806, -73.486, 67.893, 96.433, 15.421]
  MoveL 3791 to (229.48, 163.86, 59.84) mm, rotated rx -180 ry 0 rz 180 deg; joints [-67.021, 56.806, -73.486, 67.893, 96.433, 15.421]
  Call Extruder(271.01110)
  MoveL 3792 to (229.28, 163.91, 59.84) mm, rotated rx 180 ry 0 rz 180 deg; joints [-67.087, 56.803, -73.487, 67.958, 96.418, 15.433]
  MoveL 3793 to (229.28, 163.91, 59.84) mm, rotated rx 180 ry 0 rz 180 deg; joints [-67.087, 56.803, -73.487, 67.958, 96.418, 15.433]
  Call Extruder(271.12527)
  MoveL 3794 to (229.08, 163.95, 59.84) mm, rotated rx 180 ry 0 rz 180 deg; joints [-67.153, 56.8, -73.489, 68.022, 96.402, 15.444]
  MoveL 3795 to (229.08, 163.95, 59.84) mm, rotated rx 180 ry 0 rz 180 deg; joints [-67.153, 56.8, -73.489, 68.022, 96.402, 15.444]
  Call Extruder(271.23899)
  MoveL 3796 to (228.87, 164, 59.84) mm, rotated rx -180 ry 0 rz -180 deg; joints [-67.22, 56.797, -73.49, 68.087, 96.386, 15.455]
  MoveL 3797 to (228.87, 164, 59.84) mm, rotated rx -180 ry 0 rz -180 deg; joints [-67.22, 56.797, -73.49, 68.087, 96.386, 15.455]
  Call Extruder(271.36441)
  MoveL 3798 to (228.64, 164.04, 59.84) mm, rotated rx -180 ry 0 rz -180 deg; joints [-67.293, 56.794, -73.492, 68.158, 96.368, 15.468]
  MoveL 3799 to (228.64, 164.04, 59.84) mm, rotated rx -180 ry 0 rz -180 deg; joints [-67.293, 56.794, -73.492, 68.158, 96.368, 15.468]
  Call Extruder(271.50139)
  MoveL 3800 to (228.4, 164.09, 59.84) mm, rotated rx 180 ry 0 rz -180 deg; joints [-67.373, 56.79, -73.494, 68.237, 96.349, 15.482]
  MoveL 3801 to (228.4, 164.09, 59.84) mm, rotated rx 180 ry 0 rz -180 deg; joints [-67.373, 56.79, -73.494, 68.237, 96.349, 15.482]
  Call Extruder(271.63776)
  MoveL 3802 to (228.15, 164.14, 59.84) mm, rotated rx 180 ry 0 rz 180 deg; joints [-67.453, 56.786, -73.496, 68.316, 96.329, 15.496]
  MoveL 3803 to (228.15, 164.14, 59.84) mm, rotated rx 180 ry 0 rz 180 deg; joints [-67.453, 56.786, -73.496, 68.316, 96.329, 15.496]
  Call Extruder(271.77351)
  MoveL 3804 to (227.9, 164.19, 59.84) mm, rotated rx -180 ry 0 rz 180 deg; joints [-67.534, 56.782, -73.498, 68.394, 96.31, 15.51]
  MoveL 3805 to (227.9, 164.19, 59.84) mm, rotated rx -180 ry 0 rz 180 deg; joints [-67.534, 56.782, -73.498, 68.394, 96.31, 15.51]
  Call Extruder(271.90866)
  MoveL 3806 to (227.65, 164.24, 59.84) mm, rotated rx 180 ry 0 rz 180 deg; joints [-67.614, 56.779, -73.5, 68.472, 96.291, 15.524]
  MoveL 3807 to (227.65, 164.24, 59.84) mm, rotated rx 180 ry 0 rz 180 deg; joints [-67.614, 56.779, -73.5, 68.472, 96.291, 15.524]
  Call Extruder(272.04320)
  MoveL 3808 to (227.4, 164.29, 59.84) mm, rotated rx -180 ry 0 rz 180 deg; joints [-67.695, 56.775, -73.501, 68.551, 96.271, 15.538]
  MoveL 3809 to (227.4, 164.29, 59.84) mm, rotated rx -180 ry 0 rz 180 deg; joints [-67.695, 56.775, -73.501, 68.551, 96.271, 15.538]
  Call Extruder(272.17712)
  MoveL 3810 to (227.15, 164.34, 59.84) mm, rotated rx -180 ry 0 rz -180 deg; joints [-67.775, 56.771, -73.503, 68.629, 96.252, 15.551]
  MoveL 3811 to (227.15, 164.34, 59.84) mm, rotated rx -180 ry 0 rz -180 deg; joints [-67.775, 56.771, -73.503, 68.629, 96.252, 15.551]
  Call Extruder(272.32499)
  MoveL 3812 to (226.87, 164.39, 59.84) mm, rotated rx 180 ry 0 rz 180 deg; joints [-67.864, 56.767, -73.506, 68.716, 96.23, 15.567]
  MoveL 3813 to (226.87, 164.39, 59.84) mm, rotated rx 180 ry 0 rz 180 deg; joints [-67.864, 56.767, -73.506, 68.716, 96.23, 15.567]
  Call Extruder(272.48673)
  MoveL 3814 to (226.57, 164.44, 59.84) mm, rotated rx 180 ry 0 rz -180 deg; joints [-67.961, 56.761, -73.508, 68.811, 96.207, 15.585]
  MoveL 3815 to (226.57, 164.44, 59.84) mm, rotated rx 180 ry 0 rz -180 deg; joints [-67.961, 56.761, -73.508, 68.811, 96.207, 15.585]
  Call Extruder(272.64774)
  MoveL 3816 to (226.26, 164.49, 59.84) mm, rotated rx -180 ry 0 rz 180 deg; joints [-68.059, 56.756, -73.511, 68.907, 96.184, 15.603]
  MoveL 3817 to (226.26, 164.49, 59.84) mm, rotated rx -180 ry 0 rz 180 deg; joints [-68.059, 56.756, -73.511, 68.907, 96.184, 15.603]
  Call Extruder(272.80803)
  MoveL 3818 to (225.95, 164.53, 59.84) mm, rotated rx -180 ry 0 rz 180 deg; joints [-68.156, 56.751, -73.514, 69.002, 96.16, 15.62]
  MoveL 3819 to (225.95, 164.53, 59.84) mm, rotated rx -180 ry 0 rz 180 deg; joints [-68.156, 56.751, -73.514, 69.002, 96.16, 15.62]
  Call Extruder(272.96758)
  MoveL 3820 to (225.65, 164.58, 59.84) mm, rotated rx -180 ry 0 rz -180 deg; joints [-68.254, 56.745, -73.516, 69.097, 96.137, 15.638]
  MoveL 3821 to (225.65, 164.58, 59.84) mm, rotated rx -180 ry 0 rz -180 deg; joints [-68.254, 56.745, -73.516, 69.097, 96.137, 15.638]
  Call Extruder(273.12641)
  MoveL 3822 to (225.34, 164.63, 59.84) mm, rotated rx 180 ry 0 rz 180 deg; joints [-68.351, 56.74, -73.519, 69.193, 96.113, 15.656]
  MoveL 3823 to (225.34, 164.63, 59.84) mm, rotated rx 180 ry 0 rz 180 deg; joints [-68.351, 56.74, -73.519, 69.193, 96.113, 15.656]
  Call Extruder(273.30508)
  MoveL 3824 to (225, 164.68, 59.84) mm, rotated rx -180 ry 0 rz 180 deg; joints [-68.461, 56.734, -73.522, 69.3, 96.087, 15.676]
  MoveL 3825 to (225, 164.68, 59.84) mm, rotated rx -180 ry 0 rz 180 deg; joints [-68.461, 56.734, -73.522, 69.3, 96.087, 15.676]
  Call Extruder(273.50353)
  MoveL 3826 to (224.61, 164.73, 59.84) mm, rotated rx 180 ry 0 rz 180 deg; joints [-68.583, 56.726, -73.526, 69.419, 96.058, 15.699]
  MoveL 3827 to (224.61, 164.73, 59.84) mm, rotated rx 180 ry 0 rz 180 deg; joints [-68.583, 56.726, -73.526, 69.419, 96.058, 15.699]
  Call Extruder(273.70110)
  MoveL 3828 to (224.22, 164.77, 59.84) mm, rotated rx -180 ry 0 rz 180 deg; joints [-68.706, 56.718, -73.53, 69.539, 96.029, 15.722]
  MoveL 3829 to (224.22, 164.77, 59.84) mm, rotated rx -180 ry 0 rz 180 deg; joints [-68.706, 56.718, -73.53, 69.539, 96.029, 15.722]
  Call Extruder(273.89781)
  MoveL 3830 to (223.83, 164.82, 59.84) mm, rotated rx -180 ry 0 rz 180 deg; joints [-68.828, 56.711, -73.534, 69.659, 96, 15.745]
  MoveL 3831 to (223.83, 164.82, 59.84) mm, rotated rx -180 ry 0 rz 180 deg; joints [-68.828, 56.711, -73.534, 69.659, 96, 15.745]
  Call Extruder(274.09365)
  MoveL 3832 to (223.45, 164.86, 59.84) mm, rotated rx -180 ry 0 rz -180 deg; joints [-68.951, 56.703, -73.537, 69.778, 95.97, 15.769]
  MoveL 3833 to (223.45, 164.86, 59.84) mm, rotated rx -180 ry 0 rz -180 deg; joints [-68.951, 56.703, -73.537, 69.778, 95.97, 15.769]
  Call Extruder(274.38900)
  MoveL 3834 to (222.86, 164.91, 59.84) mm, rotated rx -180 ry 0 rz 180 deg; joints [-69.135, 56.69, -73.544, 69.958, 95.927, 15.805]
  MoveL 3835 to (222.86, 164.91, 59.84) mm, rotated rx -180 ry 0 rz 180 deg; joints [-69.135, 56.69, -73.544, 69.958, 95.927, 15.805]
  Call Extruder(274.68303)
  MoveL 3836 to (222.27, 164.96, 59.84) mm, rotated rx -180 ry 0 rz -180 deg; joints [-69.319, 56.678, -73.55, 70.138, 95.883, 15.842]
  MoveL 3837 to (222.27, 164.96, 59.84) mm, rotated rx -180 ry 0 rz -180 deg; joints [-69.319, 56.678, -73.55, 70.138, 95.883, 15.842]
  Call Extruder(274.97572)
  MoveL 3838 to (221.68, 165, 59.84) mm, rotated rx -180 ry 0 rz 180 deg; joints [-69.504, 56.665, -73.557, 70.319, 95.839, 15.878]
  MoveL 3839 to (221.68, 165, 59.84) mm, rotated rx -180 ry 0 rz 180 deg; joints [-69.504, 56.665, -73.557, 70.319, 95.839, 15.878]
  Call Extruder(275.54917)
  MoveL 3840 to (220.52, 165.05, 59.84) mm, rotated rx 180 ry 0 rz -180 deg; joints [-69.864, 56.637, -73.57, 70.671, 95.754, 15.952]
  MoveL 3841 to (220.52, 165.05, 59.84) mm, rotated rx 180 ry 0 rz -180 deg; joints [-69.864, 56.637, -73.57, 70.671, 95.754, 15.952]
  Call Extruder(276.26318)
  MoveL 3842 to (219.06, 165.09, 59.84) mm, rotated rx -180 ry 0 rz -180 deg; joints [-70.315, 56.602, -73.588, 71.111, 95.648, 16.046]
  Call Extruder(393.10992)
  MoveL 3843 to (-19.06, 165.09, 59.84) mm, rotated rx 180 ry 0 rz 180 deg; joints [-137.325, 61.228, -70.1, 136.981, 83.489, 6.04]
  Call Extruder(393.53852)
  MoveL 3844 to (-19.94, 165.07, 59.84) mm, rotated rx 180 ry 0 rz 180 deg; joints [-137.467, 61.265, -70.06, 137.13, 83.531, 5.971]
  MoveL 3845 to (-19.94, 165.07, 59.84) mm, rotated rx 180 ry 0 rz 180 deg; joints [-137.467, 61.265, -70.06, 137.13, 83.531, 5.971]
  Call Extruder(394.11197)
  MoveL 3846 to (-21.1, 165.03, 59.84) mm, rotated rx 180 ry 0 rz 180 deg; joints [-137.659, 61.312, -70.006, 137.329, 83.585, 5.881]
  MoveL 3847 to (-21.1, 165.03, 59.84) mm, rotated rx 180 ry 0 rz 180 deg; joints [-137.659, 61.312, -70.006, 137.329, 83.585, 5.881]
  Call Extruder(394.54627)
  MoveL 3848 to (-21.97, 164.98, 59.84) mm, rotated rx -180 ry 0 rz 180 deg; joints [-137.804, 61.347, -69.966, 137.48, 83.626, 5.813]
  MoveL 3849 to (-21.97, 164.98, 59.84) mm, rotated rx -180 ry 0 rz 180 deg; joints [-137.804, 61.347, -69.966, 137.48, 83.626, 5.813]
  Call Extruder(394.84030)
  MoveL 3850 to (-22.56, 164.93, 59.84) mm, rotated rx 180 ry 0 rz 180 deg; joints [-137.905, 61.371, -69.94, 137.585, 83.652, 5.768]
  MoveL 3851 to (-22.56, 164.93, 59.84) mm, rotated rx 180 ry 0 rz 180 deg; joints [-137.905, 61.371, -69.94, 137.585, 83.652, 5.768]
  Call Extruder(395.13566)
  MoveL 3852 to (-23.15, 164.89, 59.84) mm, rotated rx -180 ry 0 rz 180 deg; joints [-138.004, 61.394, -69.913, 137.688, 83.679, 5.723]
  MoveL 3853 to (-23.15, 164.89, 59.84) mm, rotated rx -180 ry 0 rz 180 deg; joints [-138.004, 61.394, -69.913, 137.688, 83.679, 5.723]
  Call Extruder(395.38188)
  MoveL 3854 to (-23.64, 164.84, 59.84) mm, rotated rx -180 ry 0 rz 180 deg; joints [-138.088, 61.413, -69.891, 137.775, 83.701, 5.687]
  MoveL 3855 to (-23.64, 164.84, 59.84) mm, rotated rx -180 ry 0 rz 180 deg; joints [-138.088, 61.413, -69.891, 137.775, 83.701, 5.687]
  Call Extruder(395.57858)
  MoveL 3856 to (-24.03, 164.79, 59.84) mm, rotated rx -180 ry 0 rz 180 deg; joints [-138.156, 61.427, -69.874, 137.845, 83.717, 5.658]
  MoveL 3857 to (-24.03, 164.79, 59.84) mm, rotated rx -180 ry 0 rz 180 deg; joints [-138.156, 61.427, -69.874, 137.845, 83.717, 5.658]
  Call Extruder(395.77616)
  MoveL 3858 to (-24.42, 164.75, 59.84) mm, rotated rx -180 ry 0 rz 180 deg; joints [-138.224, 61.442, -69.857, 137.916, 83.734, 5.629]
  MoveL 3859 to (-24.42, 164.75, 59.84) mm, rotated rx -180 ry 0 rz 180 deg; joints [-138.224, 61.442, -69.857, 137.916, 83.734, 5.629]
  Call Extruder(395.97460)
  MoveL 3860 to (-24.8, 164.7, 59.84) mm, rotated rx -180 ry 0 rz 180 deg; joints [-138.292, 61.456, -69.84, 137.986, 83.751, 5.6]
  MoveL 3861 to (-24.8, 164.7, 59.84) mm, rotated rx -180 ry 0 rz 180 deg; joints [-138.292, 61.456, -69.84, 137.986, 83.751, 5.6]
  Call Extruder(396.17391)
  MoveL 3862 to (-25.19, 164.66, 59.84) mm, rotated rx -180 ry 0 rz 180 deg; joints [-138.359, 61.471, -69.823, 138.056, 83.768, 5.572]
  MoveL 3863 to (-25.19, 164.66, 59.84) mm, rotated rx -180 ry 0 rz 180 deg; joints [-138.359, 61.471, -69.823, 138.056, 83.768, 5.572]
  Call Extruder(396.33274)
  MoveL 3864 to (-25.5, 164.61, 59.84) mm, rotated rx 180 ry 0 rz -180 deg; joints [-138.415, 61.482, -69.81, 138.113, 83.781, 5.55]
  MoveL 3865 to (-25.5, 164.61, 59.84) mm, rotated rx 180 ry 0 rz -180 deg; joints [-138.415, 61.482, -69.81, 138.113, 83.781, 5.55]
  Call Extruder(396.49230)
  MoveL 3866 to (-25.8, 164.56, 59.84) mm, rotated rx -180 ry 0 rz 180 deg; joints [-138.47, 61.493, -69.797, 138.17, 83.793, 5.527]
  MoveL 3867 to (-25.8, 164.56, 59.84) mm, rotated rx -180 ry 0 rz 180 deg; joints [-138.47, 61.493, -69.797, 138.17, 83.793, 5.527]
  Call Extruder(396.65259)
  MoveL 3868 to (-26.11, 164.51, 59.84) mm, rotated rx 180 ry 0 rz 180 deg; joints [-138.525, 61.504, -69.784, 138.227, 83.806, 5.505]
  MoveL 3869 to (-26.11, 164.51, 59.84) mm, rotated rx 180 ry 0 rz 180 deg; joints [-138.525, 61.504, -69.784, 138.227, 83.806, 5.505]
  Call Extruder(396.81360)
  MoveL 3870 to (-26.41, 164.46, 59.84) mm, rotated rx 180 ry 0 rz 180 deg; joints [-138.58, 61.515, -69.771, 138.284, 83.818, 5.483]
  MoveL 3871 to (-26.41, 164.46, 59.84) mm, rotated rx 180 ry 0 rz 180 deg; joints [-138.58, 61.515, -69.771, 138.284, 83.818, 5.483]
  Call Extruder(396.97535)
  MoveL 3872 to (-26.72, 164.41, 59.84) mm, rotated rx -180 ry 0 rz 180 deg; joints [-138.635, 61.527, -69.758, 138.34, 83.831, 5.461]
  MoveL 3873 to (-26.72, 164.41, 59.84) mm, rotated rx -180 ry 0 rz 180 deg; joints [-138.635, 61.527, -69.758, 138.34, 83.831, 5.461]
  Call Extruder(397.13782)
  MoveL 3874 to (-27.03, 164.37, 59.84) mm, rotated rx -180 ry 0 rz -180 deg; joints [-138.69, 61.538, -69.745, 138.397, 83.844, 5.439]
  MoveL 3875 to (-27.03, 164.37, 59.84) mm, rotated rx -180 ry 0 rz -180 deg; joints [-138.69, 61.538, -69.745, 138.397, 83.844, 5.439]
  Call Extruder(397.27175)
  MoveL 3876 to (-27.28, 164.32, 59.84) mm, rotated rx -180 ry 0 rz 180 deg; joints [-138.736, 61.546, -69.735, 138.445, 83.854, 5.421]
  MoveL 3877 to (-27.28, 164.32, 59.84) mm, rotated rx -180 ry 0 rz 180 deg; joints [-138.736, 61.546, -69.735, 138.445, 83.854, 5.421]
  Call Extruder(397.40628)
  MoveL 3878 to (-27.52, 164.27, 59.84) mm, rotated rx -180 ry 0 rz 180 deg; joints [-138.783, 61.555, -69.725, 138.493, 83.864, 5.404]
  MoveL 3879 to (-27.52, 164.27, 59.84) mm, rotated rx -180 ry 0 rz 180 deg; joints [-138.783, 61.555, -69.725, 138.493, 83.864, 5.404]
  Call Extruder(397.54143)
  MoveL 3880 to (-27.77, 164.22, 59.84) mm, rotated rx -180 ry 0 rz -180 deg; joints [-138.829, 61.564, -69.714, 138.54, 83.874, 5.386]
  MoveL 3881 to (-27.77, 164.22, 59.84) mm, rotated rx -180 ry 0 rz -180 deg; joints [-138.829, 61.564, -69.714, 138.54, 83.874, 5.386]
  Call Extruder(397.67719)
  MoveL 3882 to (-28.02, 164.17, 59.84) mm, rotated rx -180 ry 0 rz 180 deg; joints [-138.875, 61.572, -69.704, 138.588, 83.884, 5.369]
  MoveL 3883 to (-28.02, 164.17, 59.84) mm, rotated rx -180 ry 0 rz 180 deg; joints [-138.875, 61.572, -69.704, 138.588, 83.884, 5.369]
  Call Extruder(397.81355)
  MoveL 3884 to (-28.27, 164.12, 59.84) mm, rotated rx -180 ry 0 rz 180 deg; joints [-138.921, 61.581, -69.694, 138.635, 83.893, 5.351]
  MoveL 3885 to (-28.27, 164.12, 59.84) mm, rotated rx -180 ry 0 rz 180 deg; joints [-138.921, 61.581, -69.694, 138.635, 83.893, 5.351]
  Call Extruder(397.89841)
  MoveL 3886 to (-28.43, 164.09, 59.84) mm, rotated rx -180 ry 0 rz 180 deg; joints [-138.95, 61.586, -69.687, 138.665, 83.9, 5.34]
  Set speed (130.0 mm/s)
  MoveL 3887 to (-31.76, 163.31, 59.84) mm, rotated rx -180 ry 0 rz 180 deg; joints [-139.581, 61.698, -69.552, 139.314, 84.029, 5.11]
  MoveL 3888 to (-31.76, 163.31, 69.25) mm, rotated rx 180 ry 0 rz 180 deg; joints [-139.581, 63.09, -71.549, 139.271, 83.569, 5.508]
  Call Extruder(395.89841)
  Set speed (40.0 mm/s)
  MoveL 3889 to (-31.76, 163.31, 69.25) mm, rotated rx 180 ry 0 rz 180 deg; joints [-139.581, 63.09, -71.549, 139.271, 83.569, 5.508]
  Call Extruder(0.00000)
  Set speed (130.0 mm/s)
  MoveL 3890 to (-31.64, 163.21, 69.25) mm, rotated rx 180 ry 0 rz 180 deg; joints [-139.581, 63.081, -71.56, 139.27, 83.555, 5.521]
  Call Extruder(2.00000)
  Set speed (40.0 mm/s)
  MoveL 3891 to (-31.64, 163.21, 69.25) mm, rotated rx 180 ry 0 rz 180 deg; joints [-139.581, 63.081, -71.56, 139.27, 83.555, 5.521]
  Set speed (30.0 mm/s)
  MoveL 3892 to (-31.64, 163.21, 69.25) mm, rotated rx 180 ry 0 rz 180 deg; joints [-139.581, 63.081, -71.56, 139.27, 83.555, 5.521]
  Call Extruder(2.18198)
  MoveL 3893 to (-31.93, 163.09, 69.25) mm, rotated rx -180 ry 0 rz 180 deg; joints [-139.645, 63.089, -71.55, 139.335, 83.562, 5.502]
  MoveL 3894 to (-31.93, 163.09, 69.25) mm, rotated rx -180 ry 0 rz 180 deg; joints [-139.645, 63.089, -71.55, 139.335, 83.562, 5.502]
  Call Extruder(2.36471)
  MoveL 3895 to (-32.22, 162.96, 69.25) mm, rotated rx -180 ry 0 rz -180 deg; joints [-139.709, 63.097, -71.54, 139.4, 83.569, 5.483]
  MoveL 3896 to (-32.22, 162.96, 69.25) mm, rotated rx -180 ry 0 rz -180 deg; joints [-139.709, 63.097, -71.54, 139.4, 83.569, 5.483]
  Call Extruder(2.53513)
  MoveL 3897 to (-32.49, 162.85, 69.25) mm, rotated rx -180 ry 0 rz 180 deg; joints [-139.768, 63.104, -71.532, 139.461, 83.576, 5.466]
  MoveL 3898 to (-32.49, 162.85, 69.25) mm, rotated rx -180 ry 0 rz 180 deg; joints [-139.768, 63.104, -71.532, 139.461, 83.576, 5.466]
  Call Extruder(2.69310)
  MoveL 3899 to (-32.74, 162.74, 69.25) mm, rotated rx -180 ry 0 rz 180 deg; joints [-139.823, 63.111, -71.523, 139.518, 83.582, 5.45]
  MoveL 3900 to (-32.74, 162.74, 69.25) mm, rotated rx -180 ry 0 rz 180 deg; joints [-139.823, 63.111, -71.523, 139.518, 83.582, 5.45]
  Call Extruder(2.85168)
  MoveL 3901 to (-32.99, 162.64, 69.25) mm, rotated rx -180 ry 0 rz 180 deg; joints [-139.878, 63.118, -71.515, 139.574, 83.589, 5.434]
  MoveL 3902 to (-32.99, 162.64, 69.25) mm, rotated rx -180 ry 0 rz 180 deg; joints [-139.878, 63.118, -71.515, 139.574, 83.589, 5.434]
  Call Extruder(3.05784)
  MoveL 3903 to (-33.29, 162.46, 69.25) mm, rotated rx 180 ry 0 rz 180 deg; joints [-139.953, 63.125, -71.507, 139.65, 83.593, 5.416]
  MoveL 3904 to (-33.29, 162.46, 69.25) mm, rotated rx 180 ry 0 rz 180 deg; joints [-139.953, 63.125, -71.507, 139.65, 83.593, 5.416]
  Call Extruder(3.26479)
  MoveL 3905 to (-33.6, 162.29, 69.25) mm, rotated rx 180 ry 0 rz -180 deg; joints [-140.028, 63.132, -71.499, 139.726, 83.597, 5.398]
  MoveL 3906 to (-33.6, 162.29, 69.25) mm, rotated rx 180 ry 0 rz -180 deg; joints [-140.028, 63.132, -71.499, 139.726, 83.597, 5.398]
  Call Extruder(3.47251)
  MoveL 3907 to (-33.9, 162.11, 69.25) mm, rotated rx -180 ry 0 rz 180 deg; joints [-140.103, 63.138, -71.491, 139.802, 83.601, 5.38]
  MoveL 3908 to (-33.9, 162.11, 69.25) mm, rotated rx -180 ry 0 rz 180 deg; joints [-140.103, 63.138, -71.491, 139.802, 83.601, 5.38]
  Call Extruder(3.68101)
  MoveL 3909 to (-34.21, 161.94, 69.25) mm, rotated rx -180 ry 0 rz -180 deg; joints [-140.178, 63.145, -71.483, 139.878, 83.606, 5.362]
  MoveL 3910 to (-34.21, 161.94, 69.25) mm, rotated rx -180 ry 0 rz -180 deg; joints [-140.178, 63.145, -71.483, 139.878, 83.606, 5.362]
  Call Extruder(3.86055)
  MoveL 3911 to (-34.45, 161.76, 69.25) mm, rotated rx -180 ry 0 rz -180 deg; joints [-140.244, 63.149, -71.478, 139.945, 83.607, 5.348]
  MoveL 3912 to (-34.45, 161.76, 69.25) mm, rotated rx -180 ry 0 rz -180 deg; joints [-140.244, 63.149, -71.478, 139.945, 83.607, 5.348]
  Call Extruder(4.19399)
  MoveL 3913 to (-34.9, 161.43, 69.25) mm, rotated rx -180 ry 0 rz 180 deg; joints [-140.366, 63.157, -71.468, 140.069, 83.609, 5.324]
  MoveL 3914 to (-34.9, 161.43, 69.25) mm, rotated rx -180 ry 0 rz 180 deg; joints [-140.366, 63.157, -71.468, 140.069, 83.609, 5.324]
  Call Extruder(4.52861)
  MoveL 3915 to (-35.35, 161.1, 69.25) mm, rotated rx -180 ry 0 rz -180 deg; joints [-140.489, 63.165, -71.459, 140.193, 83.61, 5.299]
  Call Extruder(5.35652)
  MoveL 3916 to (-36.39, 160.19, 69.25) mm, rotated rx -180 ry 0 rz -180 deg; joints [-140.797, 63.178, -71.444, 140.503, 83.603, 5.247]
  Call Extruder(5.98652)
  MoveL 3917 to (-37.09, 159.41, 69.25) mm, rotated rx -180 ry 0 rz -180 deg; joints [-141.034, 63.18, -71.44, 140.742, 83.586, 5.216]
  Call Extruder(6.31951)
  MoveL 3918 to (-37.44, 158.97, 69.25) mm, rotated rx -180 ry 0 rz 180 deg; joints [-141.16, 63.18, -71.441, 140.868, 83.575, 5.203]
  MoveL 3919 to (-37.44, 158.97, 69.25) mm, rotated rx -180 ry 0 rz 180 deg; joints [-141.16, 63.18, -71.441, 140.868, 83.575, 5.203]
  Call Extruder(6.58931)
  MoveL 3920 to (-37.7, 158.61, 69.25) mm, rotated rx 180 ry 0 rz 180 deg; joints [-141.262, 63.179, -71.442, 140.969, 83.563, 5.193]
  Set speed (130.0 mm/s)
  MoveL 3921 to (-37.7, 158.61, 69.25) mm, rotated rx 180 ry 0 rz 180 deg; joints [-141.262, 63.179, -71.442, 140.969, 83.563, 5.193]
  Set speed (30.0 mm/s)
  MoveL 3922 to (-37.7, 158.61, 69.25) mm, rotated rx 180 ry 0 rz 180 deg; joints [-141.262, 63.179, -71.442, 140.969, 83.563, 5.193]
  Call Extruder(6.87472)
  MoveL 3923 to (-37.98, 158.22, 69.25) mm, rotated rx 180 ry 0 rz -180 deg; joints [-141.37, 63.178, -71.444, 141.078, 83.551, 5.182]
  MoveL 3924 to (-37.98, 158.22, 69.25) mm, rotated rx 180 ry 0 rz -180 deg; joints [-141.37, 63.178, -71.444, 141.078, 83.551, 5.182]
  Call Extruder(7.13432)
  MoveL 3925 to (-38.22, 157.85, 69.25) mm, rotated rx -180 ry 0 rz -180 deg; joints [-141.468, 63.175, -71.446, 141.176, 83.539, 5.174]
  MoveL 3926 to (-38.22, 157.85, 69.25) mm, rotated rx -180 ry 0 rz -180 deg; joints [-141.468, 63.175, -71.446, 141.176, 83.539, 5.174]
  Call Extruder(7.34204)
  MoveL 3927 to (-38.4, 157.55, 69.25) mm, rotated rx -180 ry 0 rz 180 deg; joints [-141.547, 63.172, -71.45, 141.254, 83.527, 5.17]
  MoveL 3928 to (-38.4, 157.55, 69.25) mm, rotated rx -180 ry 0 rz 180 deg; joints [-141.547, 63.172, -71.45, 141.254, 83.527, 5.17]
  Call Extruder(7.54898)
  MoveL 3929 to (-38.57, 157.25, 69.25) mm, rotated rx -180 ry 0 rz -180 deg; joints [-141.625, 63.17, -71.453, 141.332, 83.515, 5.165]
  MoveL 3930 to (-38.57, 157.25, 69.25) mm, rotated rx -180 ry 0 rz -180 deg; joints [-141.625, 63.17, -71.453, 141.332, 83.515, 5.165]
  Call Extruder(7.75514)
  MoveL 3931 to (-38.75, 156.94, 69.25) mm, rotated rx -180 ry 0 rz -180 deg; joints [-141.704, 63.167, -71.457, 141.411, 83.502, 5.16]
  MoveL 3932 to (-38.75, 156.94, 69.25) mm, rotated rx -180 ry 0 rz -180 deg; joints [-141.704, 63.167, -71.457, 141.411, 83.502, 5.16]
  Call Extruder(7.93681)
  MoveL 3933 to (-38.89, 156.67, 69.25) mm, rotated rx -180 ry 0 rz 180 deg; joints [-141.773, 63.163, -71.461, 141.479, 83.49, 5.157]
  MoveL 3934 to (-38.89, 156.67, 69.25) mm, rotated rx -180 ry 0 rz 180 deg; joints [-141.773, 63.163, -71.461, 141.479, 83.49, 5.157]
  Call Extruder(8.09480)
  MoveL 3935 to (-39, 156.42, 69.25) mm, rotated rx -180 ry 0 rz 180 deg; joints [-141.832, 63.159, -71.466, 141.538, 83.478, 5.155]
  MoveL 3936 to (-39, 156.42, 69.25) mm, rotated rx -180 ry 0 rz 180 deg; joints [-141.832, 63.159, -71.466, 141.538, 83.478, 5.155]
  Call Extruder(8.25218)
  MoveL 3937 to (-39.11, 156.17, 69.25) mm, rotated rx -180 ry 0 rz 180 deg; joints [-141.891, 63.155, -71.47, 141.597, 83.466, 5.154]
  MoveL 3938 to (-39.11, 156.17, 69.25) mm, rotated rx -180 ry 0 rz 180 deg; joints [-141.891, 63.155, -71.47, 141.597, 83.466, 5.154]
  Call Extruder(8.43490)
  MoveL 3939 to (-39.22, 155.87, 69.25) mm, rotated rx 180 ry 0 rz 180 deg; joints [-141.96, 63.151, -71.476, 141.665, 83.452, 5.153]
  MoveL 3940 to (-39.22, 155.87, 69.25) mm, rotated rx 180 ry 0 rz 180 deg; joints [-141.96, 63.151, -71.476, 141.665, 83.452, 5.153]
  Call Extruder(8.61686)
  MoveL 3941 to (-39.35, 155.58, 69.25) mm, rotated rx -180 ry 0 rz -180 deg; joints [-142.029, 63.146, -71.482, 141.734, 83.437, 5.151]
  MoveL 3942 to (-39.35, 155.58, 69.25) mm, rotated rx -180 ry 0 rz -180 deg; joints [-142.029, 63.146, -71.482, 141.734, 83.437, 5.151]
  Call Extruder(8.76420)
  MoveL 3943 to (-39.44, 155.34, 69.25) mm, rotated rx -180 ry 0 rz -180 deg; joints [-142.085, 63.142, -71.487, 141.789, 83.425, 5.151]
  MoveL 3944 to (-39.44, 155.34, 69.25) mm, rotated rx -180 ry 0 rz -180 deg; joints [-142.085, 63.142, -71.487, 141.789, 83.425, 5.151]
  Call Extruder(8.87743)
  MoveL 3945 to (-39.5, 155.15, 69.25) mm, rotated rx -180 ry 0 rz 180 deg; joints [-142.127, 63.138, -71.492, 141.831, 83.415, 5.151]
  MoveL 3946 to (-39.5, 155.15, 69.25) mm, rotated rx -180 ry 0 rz 180 deg; joints [-142.127, 63.138, -71.492, 141.831, 83.415, 5.151]
  Call Extruder(8.99022)
  MoveL 3947 to (-39.56, 154.97, 69.25) mm, rotated rx 180 ry 0 rz -180 deg; joints [-142.169, 63.134, -71.496, 141.872, 83.404, 5.151]
  MoveL 3948 to (-39.56, 154.97, 69.25) mm, rotated rx 180 ry 0 rz -180 deg; joints [-142.169, 63.134, -71.496, 141.872, 83.404, 5.151]
  Call Extruder(9.10257)
  MoveL 3949 to (-39.62, 154.78, 69.25) mm, rotated rx -180 ry 0 rz 180 deg; joints [-142.212, 63.13, -71.501, 141.914, 83.394, 5.152]
  MoveL 3950 to (-39.62, 154.78, 69.25) mm, rotated rx -180 ry 0 rz 180 deg; joints [-142.212, 63.13, -71.501, 141.914, 83.394, 5.152]
  Call Extruder(9.21447)
  MoveL 3951 to (-39.68, 154.59, 69.25) mm, rotated rx -180 ry 0 rz -180 deg; joints [-142.254, 63.127, -71.505, 141.956, 83.384, 5.152]
  MoveL 3952 to (-39.68, 154.59, 69.25) mm, rotated rx -180 ry 0 rz -180 deg; joints [-142.254, 63.127, -71.505, 141.956, 83.384, 5.152]
  Call Extruder(9.33587)
  MoveL 3953 to (-39.75, 154.38, 69.25) mm, rotated rx 180 ry 0 rz 180 deg; joints [-142.3, 63.122, -71.51, 142.001, 83.372, 5.152]
  MoveL 3954 to (-39.75, 154.38, 69.25) mm, rotated rx 180 ry 0 rz 180 deg; joints [-142.3, 63.122, -71.51, 142.001, 83.372, 5.152]
  Call Extruder(9.46666)
  MoveL 3955 to (-39.81, 154.16, 69.25) mm, rotated rx 180 ry 0 rz 180 deg; joints [-142.35, 63.118, -71.516, 142.05, 83.36, 5.153]
  MoveL 3956 to (-39.81, 154.16, 69.25) mm, rotated rx 180 ry 0 rz 180 deg; joints [-142.35, 63.118, -71.516, 142.05, 83.36, 5.153]
  Call Extruder(9.59689)
  MoveL 3957 to (-39.88, 153.94, 69.25) mm, rotated rx -180 ry 0 rz 180 deg; joints [-142.399, 63.113, -71.521, 142.099, 83.347, 5.154]
  MoveL 3958 to (-39.88, 153.94, 69.25) mm, rotated rx -180 ry 0 rz 180 deg; joints [-142.399, 63.113, -71.521, 142.099, 83.347, 5.154]
  Call Extruder(9.72656)
  MoveL 3959 to (-39.95, 153.71, 69.25) mm, rotated rx 180 ry 0 rz -180 deg; joints [-142.449, 63.108, -71.527, 142.148, 83.335, 5.154]
  MoveL 3960 to (-39.95, 153.71, 69.25) mm, rotated rx 180 ry 0 rz -180 deg; joints [-142.449, 63.108, -71.527, 142.148, 83.335, 5.154]
  Call Extruder(9.85565)
  MoveL 3961 to (-40.02, 153.49, 69.25) mm, rotated rx -180 ry 0 rz -180 deg; joints [-142.498, 63.104, -71.533, 142.197, 83.322, 5.155]
  MoveL 3962 to (-40.02, 153.49, 69.25) mm, rotated rx -180 ry 0 rz -180 deg; joints [-142.498, 63.104, -71.533, 142.197, 83.322, 5.155]
  Call Extruder(9.97074)
  MoveL 3963 to (-40.06, 153.28, 69.25) mm, rotated rx 180 ry 0 rz 180 deg; joints [-142.541, 63.099, -71.539, 142.24, 83.309, 5.157]
  MoveL 3964 to (-40.06, 153.28, 69.25) mm, rotated rx 180 ry 0 rz 180 deg; joints [-142.541, 63.099, -71.539, 142.24, 83.309, 5.157]
  Call Extruder(10.08538)
  MoveL 3965 to (-40.11, 153.08, 69.25) mm, rotated rx 180 ry 0 rz 180 deg; joints [-142.584, 63.094, -71.545, 142.282, 83.297, 5.158]
  MoveL 3966 to (-40.11, 153.08, 69.25) mm, rotated rx 180 ry 0 rz 180 deg; joints [-142.584, 63.094, -71.545, 142.282, 83.297, 5.158]
  Call Extruder(10.19956)
  MoveL 3967 to (-40.15, 152.88, 69.25) mm, rotated rx -180 ry 0 rz 180 deg; joints [-142.627, 63.089, -71.551, 142.324, 83.284, 5.16]
  MoveL 3968 to (-40.15, 152.88, 69.25) mm, rotated rx -180 ry 0 rz 180 deg; joints [-142.627, 63.089, -71.551, 142.324, 83.284, 5.16]
  Call Extruder(10.31329)
  MoveL 3969 to (-40.2, 152.67, 69.25) mm, rotated rx 180 ry 0 rz 180 deg; joints [-142.671, 63.084, -71.556, 142.367, 83.272, 5.162]
  MoveL 3970 to (-40.2, 152.67, 69.25) mm, rotated rx 180 ry 0 rz 180 deg; joints [-142.671, 63.084, -71.556, 142.367, 83.272, 5.162]
  Call Extruder(10.43872)
  MoveL 3971 to (-40.24, 152.44, 69.25) mm, rotated rx -180 ry 0 rz 180 deg; joints [-142.718, 63.078, -71.563, 142.414, 83.258, 5.164]
  MoveL 3972 to (-40.24, 152.44, 69.25) mm, rotated rx -180 ry 0 rz 180 deg; joints [-142.718, 63.078, -71.563, 142.414, 83.258, 5.164]
  Call Extruder(10.57569)
  MoveL 3973 to (-40.29, 152.2, 69.25) mm, rotated rx 180 ry 0 rz -180 deg; joints [-142.77, 63.072, -71.571, 142.465, 83.242, 5.166]
  MoveL 3974 to (-40.29, 152.2, 69.25) mm, rotated rx 180 ry 0 rz -180 deg; joints [-142.77, 63.072, -71.571, 142.465, 83.242, 5.166]
  Call Extruder(10.71206)
  MoveL 3975 to (-40.34, 151.95, 69.25) mm, rotated rx -180 ry 0 rz 180 deg; joints [-142.822, 63.065, -71.578, 142.516, 83.226, 5.168]
  MoveL 3976 to (-40.34, 151.95, 69.25) mm, rotated rx -180 ry 0 rz 180 deg; joints [-142.822, 63.065, -71.578, 142.516, 83.226, 5.168]
  Call Extruder(10.84781)
  MoveL 3977 to (-40.39, 151.7, 69.25) mm, rotated rx -180 ry 0 rz 180 deg; joints [-142.874, 63.059, -71.586, 142.567, 83.211, 5.171]
  MoveL 3978 to (-40.39, 151.7, 69.25) mm, rotated rx -180 ry 0 rz 180 deg; joints [-142.874, 63.059, -71.586, 142.567, 83.211, 5.171]
  Call Extruder(10.98296)
  MoveL 3979 to (-40.44, 151.45, 69.25) mm, rotated rx 180 ry 0 rz 180 deg; joints [-142.926, 63.053, -71.593, 142.619, 83.195, 5.173]
  MoveL 3980 to (-40.44, 151.45, 69.25) mm, rotated rx 180 ry 0 rz 180 deg; joints [-142.926, 63.053, -71.593, 142.619, 83.195, 5.173]
  Call Extruder(11.11749)
  MoveL 3981 to (-40.49, 151.2, 69.25) mm, rotated rx -180 ry 0 rz -180 deg; joints [-142.978, 63.046, -71.6, 142.67, 83.18, 5.175]
  MoveL 3982 to (-40.49, 151.2, 69.25) mm, rotated rx -180 ry 0 rz -180 deg; joints [-142.978, 63.046, -71.6, 142.67, 83.18, 5.175]
  Call Extruder(11.25142)
  MoveL 3983 to (-40.54, 150.95, 69.25) mm, rotated rx -180 ry 0 rz 180 deg; joints [-143.031, 63.04, -71.608, 142.721, 83.164, 5.177]
  MoveL 3984 to (-40.54, 150.95, 69.25) mm, rotated rx -180 ry 0 rz 180 deg; joints [-143.031, 63.04, -71.608, 142.721, 83.164, 5.177]
  Call Extruder(11.39927)
  MoveL 3985 to (-40.59, 150.67, 69.25) mm, rotated rx 180 ry 0 rz 180 deg; joints [-143.088, 63.033, -71.616, 142.777, 83.146, 5.18]
  MoveL 3986 to (-40.59, 150.67, 69.25) mm, rotated rx 180 ry 0 rz 180 deg; joints [-143.088, 63.033, -71.616, 142.777, 83.146, 5.18]
  Call Extruder(11.56100)
  MoveL 3987 to (-40.64, 150.37, 69.25) mm, rotated rx -180 ry 0 rz -180 deg; joints [-143.15, 63.025, -71.626, 142.839, 83.127, 5.183]
  MoveL 3988 to (-40.64, 150.37, 69.25) mm, rotated rx -180 ry 0 rz -180 deg; joints [-143.15, 63.025, -71.626, 142.839, 83.127, 5.183]
  Call Extruder(11.72199)
  MoveL 3989 to (-40.69, 150.06, 69.25) mm, rotated rx -180 ry 0 rz 180 deg; joints [-143.213, 63.016, -71.636, 142.9, 83.107, 5.187]
  MoveL 3990 to (-40.69, 150.06, 69.25) mm, rotated rx -180 ry 0 rz 180 deg; joints [-143.213, 63.016, -71.636, 142.9, 83.107, 5.187]
  Call Extruder(11.88226)
  MoveL 3991 to (-40.74, 149.76, 69.25) mm, rotated rx 180 ry 0 rz 180 deg; joints [-143.276, 63.008, -71.645, 142.962, 83.087, 5.19]
  MoveL 3992 to (-40.74, 149.76, 69.25) mm, rotated rx 180 ry 0 rz 180 deg; joints [-143.276, 63.008, -71.645, 142.962, 83.087, 5.19]
  Call Extruder(12.04180)
  MoveL 3993 to (-40.78, 149.45, 69.25) mm, rotated rx 180 ry 0 rz 180 deg; joints [-143.338, 63, -71.655, 143.024, 83.067, 5.193]
  MoveL 3994 to (-40.78, 149.45, 69.25) mm, rotated rx 180 ry 0 rz 180 deg; joints [-143.338, 63, -71.655, 143.024, 83.067, 5.193]
  Call Extruder(12.20062)
  MoveL 3995 to (-40.83, 149.14, 69.25) mm, rotated rx 180 ry 0 rz 180 deg; joints [-143.401, 62.992, -71.664, 143.085, 83.047, 5.196]
  MoveL 3996 to (-40.83, 149.14, 69.25) mm, rotated rx 180 ry 0 rz 180 deg; joints [-143.401, 62.992, -71.664, 143.085, 83.047, 5.196]
  Call Extruder(12.37928)
  MoveL 3997 to (-40.88, 148.8, 69.25) mm, rotated rx -180 ry 0 rz -180 deg; joints [-143.471, 62.982, -71.676, 143.154, 83.024, 5.2]
  MoveL 3998 to (-40.88, 148.8, 69.25) mm, rotated rx -180 ry 0 rz -180 deg; joints [-143.471, 62.982, -71.676, 143.154, 83.024, 5.2]
  Call Extruder(12.57772)
  MoveL 3999 to (-40.92, 148.41, 69.25) mm, rotated rx -180 ry 0 rz 180 deg; joints [-143.549, 62.971, -71.689, 143.23, 82.998, 5.205]
  MoveL 4000 to (-40.92, 148.41, 69.25) mm, rotated rx -180 ry 0 rz 180 deg; joints [-143.549, 62.971, -71.689, 143.23, 82.998, 5.205]
  Call Extruder(12.77530)
  MoveL 4001 to (-40.97, 148.02, 69.25) mm, rotated rx 180 ry 0 rz 180 deg; joints [-143.627, 62.96, -71.701, 143.307, 82.972, 5.21]
  MoveL 4002 to (-40.97, 148.02, 69.25) mm, rotated rx 180 ry 0 rz 180 deg; joints [-143.627, 62.96, -71.701, 143.307, 82.972, 5.21]
  Call Extruder(12.97200)
  MoveL 4003 to (-41.02, 147.63, 69.25) mm, rotated rx 180 ry 0 rz -180 deg; joints [-143.705, 62.949, -71.714, 143.383, 82.945, 5.215]
  MoveL 4004 to (-41.02, 147.63, 69.25) mm, rotated rx 180 ry 0 rz -180 deg; joints [-143.705, 62.949, -71.714, 143.383, 82.945, 5.215]
  Call Extruder(13.16784)
  MoveL 4005 to (-41.06, 147.25, 69.25) mm, rotated rx -180 ry 0 rz 180 deg; joints [-143.783, 62.938, -71.727, 143.46, 82.919, 5.219]
  MoveL 4006 to (-41.06, 147.25, 69.25) mm, rotated rx -180 ry 0 rz 180 deg; joints [-143.783, 62.938, -71.727, 143.46, 82.919, 5.219]
  Call Extruder(13.46324)
  MoveL 4007 to (-41.11, 146.66, 69.25) mm, rotated rx -180 ry 0 rz -180 deg; joints [-143.899, 62.92, -71.747, 143.573, 82.878, 5.228]
  MoveL 4008 to (-41.11, 146.66, 69.25) mm, rotated rx -180 ry 0 rz -180 deg; joints [-143.899, 62.92, -71.747, 143.573, 82.878, 5.228]
  Call Extruder(13.75731)
  MoveL 4009 to (-41.16, 146.07, 69.25) mm, rotated rx -180 ry 0 rz 180 deg; joints [-144.015, 62.903, -71.768, 143.687, 82.836, 5.236]
  MoveL 4010 to (-41.16, 146.07, 69.25) mm, rotated rx -180 ry 0 rz 180 deg; joints [-144.015, 62.903, -71.768, 143.687, 82.836, 5.236]
  Call Extruder(14.05004)
  MoveL 4011 to (-41.2, 145.48, 69.25) mm, rotated rx -180 ry 0 rz -180 deg; joints [-144.131, 62.885, -71.788, 143.801, 82.795, 5.244]
  MoveL 4012 to (-41.2, 145.48, 69.25) mm, rotated rx -180 ry 0 rz -180 deg; joints [-144.131, 62.885, -71.788, 143.801, 82.795, 5.244]
  Call Extruder(14.62350)
  MoveL 4013 to (-41.25, 144.32, 69.25) mm, rotated rx -180 ry 0 rz -180 deg; joints [-144.355, 62.848, -71.83, 144.02, 82.711, 5.263]
  MoveL 4014 to (-41.25, 144.32, 69.25) mm, rotated rx -180 ry 0 rz -180 deg; joints [-144.355, 62.848, -71.83, 144.02, 82.711, 5.263]
  Call Extruder(15.33745)
  MoveL 4015 to (-41.29, 142.86, 69.25) mm, rotated rx 180 ry 0 rz 180 deg; joints [-144.635, 62.801, -71.884, 144.293, 82.604, 5.286]
  Call Extruder(57.40228)
  MoveL 4016 to (-41.29, 57.14, 69.25) mm, rotated rx -180 ry 0 rz -180 deg; joints [-164.153, 60.402, -74.067, 163.715, 76.864, 3.798]
  Call Extruder(57.83083)
  MoveL 4017 to (-41.27, 56.26, 69.25) mm, rotated rx -180 ry 0 rz 180 deg; joints [-164.382, 60.384, -74.08, 163.948, 76.819, 3.754]
  MoveL 4018 to (-41.27, 56.26, 69.25) mm, rotated rx -180 ry 0 rz 180 deg; joints [-164.382, 60.384, -74.08, 163.948, 76.819, 3.754]
  Call Extruder(58.40429)
  MoveL 4019 to (-41.23, 55.1, 69.25) mm, rotated rx -180 ry 0 rz -180 deg; joints [-164.686, 60.36, -74.098, 164.257, 76.759, 3.694]
  MoveL 4020 to (-41.23, 55.1, 69.25) mm, rotated rx -180 ry 0 rz -180 deg; joints [-164.686, 60.36, -74.098, 164.257, 76.759, 3.694]
  Call Extruder(58.83860)
  MoveL 4021 to (-41.18, 54.23, 69.25) mm, rotated rx -180 ry 0 rz 180 deg; joints [-164.915, 60.341, -74.112, 164.49, 76.712, 3.65]
  MoveL 4022 to (-41.18, 54.23, 69.25) mm, rotated rx -180 ry 0 rz 180 deg; joints [-164.915, 60.341, -74.112, 164.49, 76.712, 3.65]
  Call Extruder(59.13267)
  MoveL 4023 to (-41.13, 53.64, 69.25) mm, rotated rx -180 ry 0 rz 180 deg; joints [-165.068, 60.327, -74.122, 164.646, 76.68, 3.62]
